        $ 3381 "bajar≔pose_add(get_actual_tcp_pose(), bajada_broca)"
        global bajar= pose_add ( get_actual_tcp_pose (), bajada_broca)
        $ 3382 "bajar" "breakAfter"
        movel(bajar, a=0.005, v=0.001)
        $ 3383 "subir≔pose_sub(get_actual_tcp_pose(), bajada_broca)"
        global subir= pose_sub ( get_actual_tcp_pose (), bajada_broca)
        $ 3384 "subir" "breakAfter"
        movel(subir, a=0.01, v=0.01)
        $ 3385 "bajada_broca≔pose_sub(bajada_broca, bajada)"
        global bajada_broca= pose_sub (bajada_broca, bajada)
        Loop_58 = Loop_58 + 1
      end
      $ 3386 "Direction: Base Z+"
      global move_thread_flag_3386=0
      thread move_thread_3386():
        enter_critical
        move_thread_flag_3386 = 1
        local towardsPos=calculate_point_to_move_towards(p[0.0,0.0,0.0,0.0,0.0,0.0], [0.0,0.0,1.0], 0.06)
        movel(towardsPos, a=0.035, v=0.03)
        move_thread_flag_3386 = 2
        exit_critical
      end
      move_thread_flag_3386 = 0
      move_thread_han_3386 = run move_thread_3386()
      while (True):
        sleep(1.0E-10)
        if (move_thread_flag_3386 > 1):
          join move_thread_han_3386
          $ 3387 "Until (distance)"
          break
        end
        sync()
      end
      $ 3388 "Set CO[1]=Apagar"
      set_configurable_digital_out(1, False)
      $ 3389 "barreno_actual≔barreno_actual+1"
      global barreno_actual=barreno_actual+1
      $ 3390 "If barreno_actual≥barrenos_menos1"
      if (barreno_actual >= barrenos_menos1):
        $ 3391 "cambiar_broca≔ True "
        global cambiar_broca=  True
      end
    end
    $ 3394 "Popup: Linea4 con chica Terminada!"
    popup("Linea4 con chica Terminada!", "Mensaje", False, False, blocking=True)
    $ 3395 "Broca_2"
    $ 3396 "Linea3"
    $ 3397 "Marcar_puntos"
    $ 3398 "MoveL"
    $ 3399 "Home3" "breakAfter"
    movel(Home3_p, a=0.5, v=0.1)
    $ 3400 "Linea3_A" "breakAfter"
    movel(Linea3_A_p, a=0.5, v=0.1)
    $ 3401 "Linea3_B" "breakAfter"
    movel(Linea3_B_p, a=0.5, v=0.1)
    $ 3402 "Linea3_C" "breakAfter"
    movel(Linea3_C_p, a=0.5, v=0.1)
    $ 3403 "Linea3_D" "breakAfter"
    movel(Linea3_D_p, a=0.5, v=0.1)
    $ 3404 "Linea3_E" "breakAfter"
    movel(Linea3_E_p, a=0.5, v=0.1)
    $ 3405 "Linea3_F" "breakAfter"
    movel(Linea3_F_p, a=0.5, v=0.1)
    $ 3406 "AB"
    $ 3407 "'desbaste_inicial'"
    # 'desbaste_inicial'
    $ 3408 "bajada_broca≔p[0,0,-0.012,0,0,0]"
    global bajada_broca=p[0,0,-0.012,0,0,0]
    $ 3409 "barrenos_menos1≔8"
    global barrenos_menos1=8
    $ 3410 "barreno_actual≔0"
    global barreno_actual=0
    $ 3411 "Loop barreno_actual≤barrenos_menos1"
    while (barreno_actual <= barrenos_menos1):
      $ 3412 "Perforacion"
      $ 3413 "MoveL"
      $ 3414 "internos≔interpolate_pose(Linea3_A, Linea3_B, barreno_actual/barrenos_menos1)"
      global internos= interpolate_pose (Linea3_A_p, Linea3_B_p, barreno_actual/barrenos_menos1)
      $ 3415 "internos" "breakAfter"
      movel(internos, a=0.5, v=0.1)
      $ 3416 "'desbaste_inicial'"
      # 'desbaste_inicial'
      $ 3417 "bajada_broca≔p[0,0,-0.012,0,0,0]"
      global bajada_broca=p[0,0,-0.012,0,0,0]
      $ 3418 "bajada≔p[0,0,0.012,0,0,0]"
      global bajada=p[0,0,0.012,0,0,0]
      $ 3419 "Direction: Base Z-"
      global move_thread_flag_3419=0
      thread move_thread_3419():
        enter_critical
        move_thread_flag_3419 = 1
        local towardsPos=calculate_point_to_move_towards(p[0.0,0.0,0.0,0.0,0.0,0.0], [0.0,0.0,-1.0], 0.076)
        movel(towardsPos, a=0.015, v=0.02)
        move_thread_flag_3419 = 2
        exit_critical
      end
      move_thread_flag_3419 = 0
      move_thread_han_3419 = run move_thread_3419()
      while (True):
        sleep(1.0E-10)
        if (move_thread_flag_3419 > 1):
          join move_thread_han_3419
          $ 3420 "Until (distance)"
          break
        end
        sync()
      end
      $ 3421 "Popup: punto contacto alanzdo"
      popup("punto contacto alanzdo", "Mensaje", False, False, blocking=True)
      $ 3422 "Direction: Base Z+"
      global move_thread_flag_3422=0
      thread move_thread_3422():
        enter_critical
        move_thread_flag_3422 = 1
        local towardsPos=calculate_point_to_move_towards(p[0.0,0.0,0.0,0.0,0.0,0.0], [0.0,0.0,1.0], 0.002)
        movel(towardsPos, a=0.005, v=0.003)
        move_thread_flag_3422 = 2
        exit_critical
      end
      move_thread_flag_3422 = 0
      move_thread_han_3422 = run move_thread_3422()
      while (True):
        sleep(1.0E-10)
        if (move_thread_flag_3422 > 1):
          join move_thread_han_3422
          $ 3423 "Until (distance)"
          break
        end
        sync()
      end
      $ 3424 "Wait: 0.3"
      sleep(0.3)
      $ 3425 "Set CO[1]=Encender"
      set_configurable_digital_out(1, True)
      $ 3426 "Wait: 0.3"
      sleep(0.3)
      $ 3427 "Loop 2 times"
      Loop_60 = 0
      while (Loop_60 < 2):
        $ 3428 "bajar≔pose_add(get_actual_tcp_pose(), bajada_broca)"
        global bajar= pose_add ( get_actual_tcp_pose (), bajada_broca)
        $ 3429 "bajar" "breakAfter"
        movel(bajar, a=0.005, v=0.001)
        $ 3430 "subir≔pose_sub(get_actual_tcp_pose(), bajada_broca)"
        global subir= pose_sub ( get_actual_tcp_pose (), bajada_broca)
        $ 3431 "subir" "breakAfter"
        movel(subir, a=0.01, v=0.01)
        $ 3432 "bajada_broca≔pose_sub(bajada_broca, bajada)"
        global bajada_broca= pose_sub (bajada_broca, bajada)
        Loop_60 = Loop_60 + 1
      end
      $ 3433 "Direction: Base Z+"
      global move_thread_flag_3433=0
      thread move_thread_3433():
        enter_critical
        move_thread_flag_3433 = 1
        local towardsPos=calculate_point_to_move_towards(p[0.0,0.0,0.0,0.0,0.0,0.0], [0.0,0.0,1.0], 0.06)
        movel(towardsPos, a=0.035, v=0.03)
        move_thread_flag_3433 = 2
        exit_critical
      end
      move_thread_flag_3433 = 0
      move_thread_han_3433 = run move_thread_3433()
      while (True):
        sleep(1.0E-10)
        if (move_thread_flag_3433 > 1):
          join move_thread_han_3433
          $ 3434 "Until (distance)"
          break
        end
        sync()
      end
      $ 3435 "Set CO[1]=Apagar"
      set_configurable_digital_out(1, False)
      $ 3436 "barreno_actual≔barreno_actual+1"
      global barreno_actual=barreno_actual+1
    end
    $ 3439 "CD"
    $ 3440 "'desbaste_inicial'"
    # 'desbaste_inicial'
    $ 3441 "bajada_broca≔p[0,0,-0.012,0,0,0]"
    global bajada_broca=p[0,0,-0.012,0,0,0]
    $ 3442 "barrenos_menos1≔8"
    global barrenos_menos1=8
    $ 3443 "barreno_actual≔0"
    global barreno_actual=0
    $ 3444 "Loop barreno_actual≤barrenos_menos1"
    while (barreno_actual <= barrenos_menos1):
      $ 3445 "Perforacion"
      $ 3446 "MoveL"
      $ 3447 "internos≔interpolate_pose(Linea3_C, Linea3_D, barreno_actual/barrenos_menos1)"
      global internos= interpolate_pose (Linea3_C_p, Linea3_D_p, barreno_actual/barrenos_menos1)
      $ 3448 "internos" "breakAfter"
      movel(internos, a=0.5, v=0.1)
      $ 3449 "'desbaste_inicial'"
      # 'desbaste_inicial'
      $ 3450 "bajada_broca≔p[0,0,-0.012,0,0,0]"
      global bajada_broca=p[0,0,-0.012,0,0,0]
      $ 3451 "bajada≔p[0,0,0.012,0,0,0]"
      global bajada=p[0,0,0.012,0,0,0]
      $ 3452 "Direction: Base Z-"
      global move_thread_flag_3452=0
      thread move_thread_3452():
        enter_critical
        move_thread_flag_3452 = 1
        local towardsPos=calculate_point_to_move_towards(p[0.0,0.0,0.0,0.0,0.0,0.0], [0.0,0.0,-1.0], 0.076)
        movel(towardsPos, a=0.015, v=0.02)
        move_thread_flag_3452 = 2
        exit_critical
      end
      move_thread_flag_3452 = 0
      move_thread_han_3452 = run move_thread_3452()
      while (True):
        sleep(1.0E-10)
        if (move_thread_flag_3452 > 1):
          join move_thread_han_3452
          $ 3453 "Until (distance)"
          break
        end
        sync()
      end
      $ 3454 "Popup: punto contacto alanzdo"
      popup("punto contacto alanzdo", "Mensaje", False, False, blocking=True)
      $ 3455 "Direction: Base Z+"
      global move_thread_flag_3455=0
      thread move_thread_3455():
        enter_critical
        move_thread_flag_3455 = 1
        local towardsPos=calculate_point_to_move_towards(p[0.0,0.0,0.0,0.0,0.0,0.0], [0.0,0.0,1.0], 0.002)
        movel(towardsPos, a=0.005, v=0.003)
        move_thread_flag_3455 = 2
        exit_critical
      end
      move_thread_flag_3455 = 0
      move_thread_han_3455 = run move_thread_3455()
      while (True):
        sleep(1.0E-10)
        if (move_thread_flag_3455 > 1):
          join move_thread_han_3455
          $ 3456 "Until (distance)"
          break
        end
        sync()
      end
      $ 3457 "Wait: 0.3"
      sleep(0.3)
      $ 3458 "Set CO[1]=Encender"
      set_configurable_digital_out(1, True)
      $ 3459 "Wait: 0.3"
      sleep(0.3)
      $ 3460 "Loop 2 times"
      Loop_64 = 0
      while (Loop_64 < 2):
        $ 3461 "bajar≔pose_add(get_actual_tcp_pose(), bajada_broca)"
        global bajar= pose_add ( get_actual_tcp_pose (), bajada_broca)
        $ 3462 "bajar" "breakAfter"
        movel(bajar, a=0.005, v=0.001)
        $ 3463 "subir≔pose_sub(get_actual_tcp_pose(), bajada_broca)"
        global subir= pose_sub ( get_actual_tcp_pose (), bajada_broca)
        $ 3464 "subir" "breakAfter"
        movel(subir, a=0.01, v=0.01)
        $ 3465 "bajada_broca≔pose_sub(bajada_broca, bajada)"
        global bajada_broca= pose_sub (bajada_broca, bajada)
        Loop_64 = Loop_64 + 1
      end
      $ 3466 "Direction: Base Z+"
      global move_thread_flag_3466=0
      thread move_thread_3466():
        enter_critical
        move_thread_flag_3466 = 1
        local towardsPos=calculate_point_to_move_towards(p[0.0,0.0,0.0,0.0,0.0,0.0], [0.0,0.0,1.0], 0.06)
        movel(towardsPos, a=0.035, v=0.03)
        move_thread_flag_3466 = 2
        exit_critical
      end
      move_thread_flag_3466 = 0
      move_thread_han_3466 = run move_thread_3466()
      while (True):
        sleep(1.0E-10)
        if (move_thread_flag_3466 > 1):
          join move_thread_han_3466
          $ 3467 "Until (distance)"
          break
        end
        sync()
      end
      $ 3468 "Set CO[1]=Apagar"
      set_configurable_digital_out(1, False)
      $ 3469 "barreno_actual≔barreno_actual+1"
      global barreno_actual=barreno_actual+1
    end
    $ 3472 "EF"
    $ 3473 "'desbaste_inicial'"
    # 'desbaste_inicial'
    $ 3474 "bajada_broca≔p[0,0,-0.012,0,0,0]"
    global bajada_broca=p[0,0,-0.012,0,0,0]
    $ 3475 "barrenos_menos1≔8"
    global barrenos_menos1=8
    $ 3476 "barreno_actual≔0"
    global barreno_actual=0
    $ 3477 "Loop barreno_actual≤barrenos_menos1"
    while (barreno_actual <= barrenos_menos1):
      $ 3478 "Perforacion"
      $ 3479 "MoveL"
      $ 3480 "internos≔interpolate_pose(Linea3_E, Linea3_F, barreno_actual/barrenos_menos1)"
      global internos= interpolate_pose (Linea3_E_p, Linea3_F_p, barreno_actual/barrenos_menos1)
      $ 3481 "internos" "breakAfter"
      movel(internos, a=0.5, v=0.1)
      $ 3482 "'desbaste_inicial'"
      # 'desbaste_inicial'
      $ 3483 "bajada_broca≔p[0,0,-0.012,0,0,0]"
      global bajada_broca=p[0,0,-0.012,0,0,0]
      $ 3484 "bajada≔p[0,0,0.012,0,0,0]"
      global bajada=p[0,0,0.012,0,0,0]
      $ 3485 "Direction: Base Z-"
      global move_thread_flag_3485=0
      thread move_thread_3485():
        enter_critical
        move_thread_flag_3485 = 1
        local towardsPos=calculate_point_to_move_towards(p[0.0,0.0,0.0,0.0,0.0,0.0], [0.0,0.0,-1.0], 0.076)
        movel(towardsPos, a=0.015, v=0.02)
        move_thread_flag_3485 = 2
        exit_critical
      end
      move_thread_flag_3485 = 0
      move_thread_han_3485 = run move_thread_3485()
      while (True):
        sleep(1.0E-10)
        if (move_thread_flag_3485 > 1):
          join move_thread_han_3485
          $ 3486 "Until (distance)"
          break
        end
        sync()
      end
      $ 3487 "Popup: punto contacto alanzdo"
      popup("punto contacto alanzdo", "Mensaje", False, False, blocking=True)
      $ 3488 "Direction: Base Z+"
      global move_thread_flag_3488=0
      thread move_thread_3488():
        enter_critical
        move_thread_flag_3488 = 1
        local towardsPos=calculate_point_to_move_towards(p[0.0,0.0,0.0,0.0,0.0,0.0], [0.0,0.0,1.0], 0.002)
        movel(towardsPos, a=0.005, v=0.003)
        move_thread_flag_3488 = 2
        exit_critical
      end
      move_thread_flag_3488 = 0
      move_thread_han_3488 = run move_thread_3488()
      while (True):
        sleep(1.0E-10)
        if (move_thread_flag_3488 > 1):
          join move_thread_han_3488
          $ 3489 "Until (distance)"
          break
        end
        sync()
      end
      $ 3490 "Wait: 0.3"
      sleep(0.3)
      $ 3491 "Set CO[1]=Encender"
      set_configurable_digital_out(1, True)
      $ 3492 "Wait: 0.3"
      sleep(0.3)
      $ 3493 "Loop 2 times"
      Loop_68 = 0
      while (Loop_68 < 2):
        $ 3494 "bajar≔pose_add(get_actual_tcp_pose(), bajada_broca)"
        global bajar= pose_add ( get_actual_tcp_pose (), bajada_broca)
        $ 3495 "bajar" "breakAfter"
        movel(bajar, a=0.005, v=0.001)
        $ 3496 "subir≔pose_sub(get_actual_tcp_pose(), bajada_broca)"
        global subir= pose_sub ( get_actual_tcp_pose (), bajada_broca)
        $ 3497 "subir" "breakAfter"
        movel(subir, a=0.01, v=0.01)
        $ 3498 "bajada_broca≔pose_sub(bajada_broca, bajada)"
        global bajada_broca= pose_sub (bajada_broca, bajada)
        Loop_68 = Loop_68 + 1
      end
      $ 3499 "Direction: Base Z+"
      global move_thread_flag_3499=0
      thread move_thread_3499():
        enter_critical
        move_thread_flag_3499 = 1
        local towardsPos=calculate_point_to_move_towards(p[0.0,0.0,0.0,0.0,0.0,0.0], [0.0,0.0,1.0], 0.06)
        movel(towardsPos, a=0.035, v=0.03)
        move_thread_flag_3499 = 2
        exit_critical
      end
      move_thread_flag_3499 = 0
      move_thread_han_3499 = run move_thread_3499()
      while (True):
        sleep(1.0E-10)
        if (move_thread_flag_3499 > 1):
          join move_thread_han_3499
          $ 3500 "Until (distance)"
          break
        end
        sync()
      end
      $ 3501 "Set CO[1]=Apagar"
      set_configurable_digital_out(1, False)
      $ 3502 "barreno_actual≔barreno_actual+1"
      global barreno_actual=barreno_actual+1
    end
    $ 3505 "Popup: Linea3 con media Terminada!"
    popup("Linea3 con media Terminada!", "Mensaje", False, False, blocking=True)
    $ 3506 "Linea4"
    $ 3507 "Marcar_puntos"
    $ 3508 "MoveL"
    $ 3509 "Home3" "breakAfter"
    movel(Home3_p, a=0.5, v=0.1)
    $ 3510 "Linea4_A" "breakAfter"
    movel(Linea4_A_p, a=0.5, v=0.1)
    $ 3511 "Linea4_B" "breakAfter"
    movel(Linea4_B_p, a=0.5, v=0.1)
    $ 3512 "Linea4_C" "breakAfter"
    movel(Linea4_C_p, a=0.5, v=0.1)
    $ 3513 "Linea4_D" "breakAfter"
    movel(Linea4_D_p, a=0.5, v=0.1)
    $ 3514 "Linea4_E" "breakAfter"
    movel(Linea4_E_p, a=0.5, v=0.1)
    $ 3515 "Linea4_F" "breakAfter"
    movel(Linea4_F_p, a=0.5, v=0.1)
    $ 3516 "AB"
    $ 3517 "'desbaste_inicial'"
    # 'desbaste_inicial'
    $ 3518 "bajada_broca≔p[0,0,-0.012,0,0,0]"
    global bajada_broca=p[0,0,-0.012,0,0,0]
    $ 3519 "barrenos_menos1≔8"
    global barrenos_menos1=8
    $ 3520 "barreno_actual≔0"
    global barreno_actual=0
    $ 3521 "Loop barreno_actual≤barrenos_menos1"
    while (barreno_actual <= barrenos_menos1):
      $ 3522 "Perforacion"
      $ 3523 "MoveL"
      $ 3524 "internos≔interpolate_pose(Linea4_A, Linea4_B, barreno_actual/barrenos_menos1)"
      global internos= interpolate_pose (Linea4_A_p, Linea4_B_p, barreno_actual/barrenos_menos1)
      $ 3525 "internos" "breakAfter"
      movel(internos, a=0.5, v=0.1)
      $ 3526 "'desbaste_inicial'"
      # 'desbaste_inicial'
      $ 3527 "bajada_broca≔p[0,0,-0.012,0,0,0]"
      global bajada_broca=p[0,0,-0.012,0,0,0]
      $ 3528 "bajada≔p[0,0,0.012,0,0,0]"
      global bajada=p[0,0,0.012,0,0,0]
      $ 3529 "Direction: Base Z-"
      global move_thread_flag_3529=0
      thread move_thread_3529():
        enter_critical
        move_thread_flag_3529 = 1
        local towardsPos=calculate_point_to_move_towards(p[0.0,0.0,0.0,0.0,0.0,0.0], [0.0,0.0,-1.0], 0.073)
        movel(towardsPos, a=0.015, v=0.02)
        move_thread_flag_3529 = 2
        exit_critical
      end
      move_thread_flag_3529 = 0
      move_thread_han_3529 = run move_thread_3529()
      while (True):
        sleep(1.0E-10)
        if (move_thread_flag_3529 > 1):
          join move_thread_han_3529
          $ 3530 "Until (distance)"
          break
        end
        sync()
      end
      $ 3531 "Popup: punto contacto alanzdo"
      popup("punto contacto alanzdo", "Mensaje", False, False, blocking=True)
      $ 3532 "Direction: Base Z+"
      global move_thread_flag_3532=0
      thread move_thread_3532():
        enter_critical
        move_thread_flag_3532 = 1
        local towardsPos=calculate_point_to_move_towards(p[0.0,0.0,0.0,0.0,0.0,0.0], [0.0,0.0,1.0], 0.002)
        movel(towardsPos, a=0.005, v=0.003)
        move_thread_flag_3532 = 2
        exit_critical
      end
      move_thread_flag_3532 = 0
      move_thread_han_3532 = run move_thread_3532()
      while (True):
        sleep(1.0E-10)
        if (move_thread_flag_3532 > 1):
          join move_thread_han_3532
          $ 3533 "Until (distance)"
          break
        end
        sync()
      end
      $ 3534 "Wait: 0.3"
      sleep(0.3)
      $ 3535 "Set CO[1]=Encender"
      set_configurable_digital_out(1, True)
      $ 3536 "Wait: 0.3"
      sleep(0.3)
      $ 3537 "Loop 2 times"
      Loop_72 = 0
      while (Loop_72 < 2):
        $ 3538 "bajar≔pose_add(get_actual_tcp_pose(), bajada_broca)"
        global bajar= pose_add ( get_actual_tcp_pose (), bajada_broca)
        $ 3539 "bajar" "breakAfter"
        movel(bajar, a=0.005, v=0.001)
        $ 3540 "subir≔pose_sub(get_actual_tcp_pose(), bajada_broca)"
        global subir= pose_sub ( get_actual_tcp_pose (), bajada_broca)
        $ 3541 "subir" "breakAfter"
        movel(subir, a=0.01, v=0.01)
        $ 3542 "bajada_broca≔pose_sub(bajada_broca, bajada)"
        global bajada_broca= pose_sub (bajada_broca, bajada)
        Loop_72 = Loop_72 + 1
      end
      $ 3543 "Direction: Base Z+"
      global move_thread_flag_3543=0
      thread move_thread_3543():
        enter_critical
        move_thread_flag_3543 = 1
        local towardsPos=calculate_point_to_move_towards(p[0.0,0.0,0.0,0.0,0.0,0.0], [0.0,0.0,1.0], 0.06)
        movel(towardsPos, a=0.035, v=0.03)
        move_thread_flag_3543 = 2
        exit_critical
      end
      move_thread_flag_3543 = 0
      move_thread_han_3543 = run move_thread_3543()
      while (True):
        sleep(1.0E-10)
        if (move_thread_flag_3543 > 1):
          join move_thread_han_3543
          $ 3544 "Until (distance)"
          break
        end
        sync()
      end
      $ 3545 "Set CO[1]=Apagar"
      set_configurable_digital_out(1, False)
      $ 3546 "barreno_actual≔barreno_actual+1"
      global barreno_actual=barreno_actual+1
    end
    $ 3549 "CD"
    $ 3550 "'desbaste_inicial'"
    # 'desbaste_inicial'
    $ 3551 "bajada_broca≔p[0,0,-0.012,0,0,0]"
    global bajada_broca=p[0,0,-0.012,0,0,0]
    $ 3552 "barrenos_menos1≔8"
    global barrenos_menos1=8
    $ 3553 "barreno_actual≔0"
    global barreno_actual=0
    $ 3554 "Loop barreno_actual≤barrenos_menos1"
    while (barreno_actual <= barrenos_menos1):
      $ 3555 "Perforacion"
      $ 3556 "MoveL"
      $ 3557 "internos≔interpolate_pose(Linea4_C, Linea4_D, barreno_actual/barrenos_menos1)"
      global internos= interpolate_pose (Linea4_C_p, Linea4_D_p, barreno_actual/barrenos_menos1)
      $ 3558 "internos" "breakAfter"
      movel(internos, a=0.5, v=0.1)
      $ 3559 "'desbaste_inicial'"
      # 'desbaste_inicial'
      $ 3560 "bajada_broca≔p[0,0,-0.012,0,0,0]"
      global bajada_broca=p[0,0,-0.012,0,0,0]
      $ 3561 "bajada≔p[0,0,0.012,0,0,0]"
      global bajada=p[0,0,0.012,0,0,0]
      $ 3562 "Direction: Base Z-"
      global move_thread_flag_3562=0
      thread move_thread_3562():
        enter_critical
        move_thread_flag_3562 = 1
        local towardsPos=calculate_point_to_move_towards(p[0.0,0.0,0.0,0.0,0.0,0.0], [0.0,0.0,-1.0], 0.073)
        movel(towardsPos, a=0.015, v=0.02)
        move_thread_flag_3562 = 2
        exit_critical
      end
      move_thread_flag_3562 = 0
      move_thread_han_3562 = run move_thread_3562()
      while (True):
        sleep(1.0E-10)
        if (move_thread_flag_3562 > 1):
          join move_thread_han_3562
          $ 3563 "Until (distance)"
          break
        end
        sync()
      end
      $ 3564 "Popup: punto contacto alanzdo"
      popup("punto contacto alanzdo", "Mensaje", False, False, blocking=True)
      $ 3565 "Direction: Base Z+"
      global move_thread_flag_3565=0
      thread move_thread_3565():
        enter_critical
        move_thread_flag_3565 = 1
        local towardsPos=calculate_point_to_move_towards(p[0.0,0.0,0.0,0.0,0.0,0.0], [0.0,0.0,1.0], 0.002)
        movel(towardsPos, a=0.005, v=0.003)
        move_thread_flag_3565 = 2
        exit_critical
      end
      move_thread_flag_3565 = 0
      move_thread_han_3565 = run move_thread_3565()
      while (True):
        sleep(1.0E-10)
        if (move_thread_flag_3565 > 1):
          join move_thread_han_3565
          $ 3566 "Until (distance)"
          break
        end
        sync()
      end
      $ 3567 "Wait: 0.3"
      sleep(0.3)
      $ 3568 "Set CO[1]=Encender"
      set_configurable_digital_out(1, True)
      $ 3569 "Wait: 0.3"
      sleep(0.3)
      $ 3570 "Loop 2 times"
      Loop_77 = 0
      while (Loop_77 < 2):
        $ 3571 "bajar≔pose_add(get_actual_tcp_pose(), bajada_broca)"
        global bajar= pose_add ( get_actual_tcp_pose (), bajada_broca)
        $ 3572 "bajar" "breakAfter"
        movel(bajar, a=0.005, v=0.001)
        $ 3573 "subir≔pose_sub(get_actual_tcp_pose(), bajada_broca)"
        global subir= pose_sub ( get_actual_tcp_pose (), bajada_broca)
        $ 3574 "subir" "breakAfter"
        movel(subir, a=0.01, v=0.01)
        $ 3575 "bajada_broca≔pose_sub(bajada_broca, bajada)"
        global bajada_broca= pose_sub (bajada_broca, bajada)
        Loop_77 = Loop_77 + 1
      end
      $ 3576 "Direction: Base Z+"
      global move_thread_flag_3576=0
      thread move_thread_3576():
        enter_critical
        move_thread_flag_3576 = 1
        local towardsPos=calculate_point_to_move_towards(p[0.0,0.0,0.0,0.0,0.0,0.0], [0.0,0.0,1.0], 0.06)
        movel(towardsPos, a=0.035, v=0.03)
        move_thread_flag_3576 = 2
        exit_critical
      end
      move_thread_flag_3576 = 0
      move_thread_han_3576 = run move_thread_3576()
      while (True):
        sleep(1.0E-10)
        if (move_thread_flag_3576 > 1):
          join move_thread_han_3576
          $ 3577 "Until (distance)"
          break
        end
        sync()
      end
      $ 3578 "Set CO[1]=Apagar"
      set_configurable_digital_out(1, False)
      $ 3579 "barreno_actual≔barreno_actual+1"
      global barreno_actual=barreno_actual+1
    end
    $ 3582 "EF"
    $ 3583 "'desbaste_inicial'"
    # 'desbaste_inicial'
    $ 3584 "bajada_broca≔p[0,0,-0.012,0,0,0]"
    global bajada_broca=p[0,0,-0.012,0,0,0]
    $ 3585 "barrenos_menos1≔8"
    global barrenos_menos1=8
    $ 3586 "barreno_actual≔0"
    global barreno_actual=0
    $ 3587 "Loop barreno_actual≤barrenos_menos1"
    while (barreno_actual <= barrenos_menos1):
      $ 3588 "Perforacion"
      $ 3589 "MoveL"
      $ 3590 "internos≔interpolate_pose(Linea4_E, Linea4_F, barreno_actual/barrenos_menos1)"
      global internos= interpolate_pose (Linea4_E_p, Linea4_F_p, barreno_actual/barrenos_menos1)
      $ 3591 "internos" "breakAfter"
      movel(internos, a=0.5, v=0.1)
      $ 3592 "'desbaste_inicial'"
      # 'desbaste_inicial'
      $ 3593 "bajada_broca≔p[0,0,-0.012,0,0,0]"
      global bajada_broca=p[0,0,-0.012,0,0,0]
      $ 3594 "bajada≔p[0,0,0.012,0,0,0]"
      global bajada=p[0,0,0.012,0,0,0]
      $ 3595 "Direction: Base Z-"
      global move_thread_flag_3595=0
      thread move_thread_3595():
        enter_critical
        move_thread_flag_3595 = 1
        local towardsPos=calculate_point_to_move_towards(p[0.0,0.0,0.0,0.0,0.0,0.0], [0.0,0.0,-1.0], 0.073)
        movel(towardsPos, a=0.015, v=0.02)
        move_thread_flag_3595 = 2
        exit_critical
      end
      move_thread_flag_3595 = 0
      move_thread_han_3595 = run move_thread_3595()
      while (True):
        sleep(1.0E-10)
        if (move_thread_flag_3595 > 1):
          join move_thread_han_3595
          $ 3596 "Until (distance)"
          break
        end
        sync()
      end
      $ 3597 "Popup: punto contacto alanzdo"
      popup("punto contacto alanzdo", "Mensaje", False, False, blocking=True)
      $ 3598 "Direction: Base Z+"
      global move_thread_flag_3598=0
      thread move_thread_3598():
        enter_critical
        move_thread_flag_3598 = 1
        local towardsPos=calculate_point_to_move_towards(p[0.0,0.0,0.0,0.0,0.0,0.0], [0.0,0.0,1.0], 0.002)
        movel(towardsPos, a=0.005, v=0.003)
        move_thread_flag_3598 = 2
        exit_critical
      end
      move_thread_flag_3598 = 0
      move_thread_han_3598 = run move_thread_3598()
      while (True):
        sleep(1.0E-10)
        if (move_thread_flag_3598 > 1):
          join move_thread_han_3598
          $ 3599 "Until (distance)"
          break
        end
        sync()
      end
      $ 3600 "Wait: 0.3"
      sleep(0.3)
      $ 3601 "Set CO[1]=Encender"
      set_configurable_digital_out(1, True)
      $ 3602 "Wait: 0.3"
      sleep(0.3)
      $ 3603 "Loop 2 times"
      Loop_81 = 0
      while (Loop_81 < 2):
        $ 3604 "bajar≔pose_add(get_actual_tcp_pose(), bajada_broca)"
        global bajar= pose_add ( get_actual_tcp_pose (), bajada_broca)
        $ 3605 "bajar" "breakAfter"
        movel(bajar, a=0.005, v=0.001)
        $ 3606 "subir≔pose_sub(get_actual_tcp_pose(), bajada_broca)"
        global subir= pose_sub ( get_actual_tcp_pose (), bajada_broca)
        $ 3607 "subir" "breakAfter"
        movel(subir, a=0.01, v=0.01)
        $ 3608 "bajada_broca≔pose_sub(bajada_broca, bajada)"
        global bajada_broca= pose_sub (bajada_broca, bajada)
        Loop_81 = Loop_81 + 1
      end
      $ 3609 "Direction: Base Z+"
      global move_thread_flag_3609=0
      thread move_thread_3609():
        enter_critical
        move_thread_flag_3609 = 1
        local towardsPos=calculate_point_to_move_towards(p[0.0,0.0,0.0,0.0,0.0,0.0], [0.0,0.0,1.0], 0.06)
        movel(towardsPos, a=0.035, v=0.03)
        move_thread_flag_3609 = 2
        exit_critical
      end
      move_thread_flag_3609 = 0
      move_thread_han_3609 = run move_thread_3609()
      while (True):
        sleep(1.0E-10)
        if (move_thread_flag_3609 > 1):
          join move_thread_han_3609
          $ 3610 "Until (distance)"
          break
        end
        sync()
      end
      $ 3611 "Set CO[1]=Apagar"
      set_configurable_digital_out(1, False)
      $ 3612 "barreno_actual≔barreno_actual+1"
      global barreno_actual=barreno_actual+1
      $ 3613 "If barreno_actual≥barrenos_menos1"
      if (barreno_actual >= barrenos_menos1):
        $ 3614 "cambiar_broca≔ True "
        global cambiar_broca=  True
      end
    end
    $ 3617 "Popup: Linea4 con media Terminada!"
    popup("Linea4 con media Terminada!", "Mensaje", False, False, blocking=True)
    $ 3618 "Broca_3"
    $ 3619 "Linea3"
    $ 3620 "Marcar_puntos"
    $ 3621 "MoveL"
    $ 3622 "Home3" "breakAfter"
    movel(Home3_p, a=0.5, v=0.1)
    $ 3623 "Linea3_A" "breakAfter"
    movel(Linea3_A_p, a=0.5, v=0.1)
    $ 3624 "Linea3_B" "breakAfter"
    movel(Linea3_B_p, a=0.5, v=0.1)
    $ 3625 "Linea3_C" "breakAfter"
    movel(Linea3_C_p, a=0.5, v=0.1)
    $ 3626 "Linea3_D" "breakAfter"
    movel(Linea3_D_p, a=0.5, v=0.1)
    $ 3627 "Linea3_E" "breakAfter"
    movel(Linea3_E_p, a=0.5, v=0.1)
    $ 3628 "Linea3_F" "breakAfter"
    movel(Linea3_F_p, a=0.5, v=0.1)
    $ 3629 "AB"
    $ 3630 "'desbaste_inicial'"
    # 'desbaste_inicial'
    $ 3631 "bajada_broca≔p[0,0,-0.024,0,0,0]"
    global bajada_broca=p[0,0,-0.024,0,0,0]
    $ 3632 "barrenos_menos1≔8"
    global barrenos_menos1=8
    $ 3633 "barreno_actual≔0"
    global barreno_actual=0
    $ 3634 "Loop barreno_actual≤barrenos_menos1"
    while (barreno_actual <= barrenos_menos1):
      $ 3635 "Perforacion"
      $ 3636 "MoveL"
      $ 3637 "internos≔interpolate_pose(Linea3_A, Linea3_B, barreno_actual/barrenos_menos1)"
      global internos= interpolate_pose (Linea3_A_p, Linea3_B_p, barreno_actual/barrenos_menos1)
      $ 3638 "internos" "breakAfter"
      movel(internos, a=0.5, v=0.1)
      $ 3639 "'desbaste_inicial'"
      # 'desbaste_inicial'
      $ 3640 "bajada_broca≔p[0,0,-0.024,0,0,0]"
      global bajada_broca=p[0,0,-0.024,0,0,0]
      $ 3641 "bajada≔p[0,0,0.024,0,0,0]"
      global bajada=p[0,0,0.024,0,0,0]
      $ 3642 "Direction: Base Z-"
      global move_thread_flag_3642=0
      thread move_thread_3642():
        enter_critical
        move_thread_flag_3642 = 1
        local towardsPos=calculate_point_to_move_towards(p[0.0,0.0,0.0,0.0,0.0,0.0], [0.0,0.0,-1.0], 0.076)
        movel(towardsPos, a=0.015, v=0.02)
        move_thread_flag_3642 = 2
        exit_critical
      end
      move_thread_flag_3642 = 0
      move_thread_han_3642 = run move_thread_3642()
      while (True):
        sleep(1.0E-10)
        if (move_thread_flag_3642 > 1):
          join move_thread_han_3642
          $ 3643 "Until (distance)"
          break
        end
        sync()
      end
      $ 3644 "Popup: punto contacto alanzdo"
      popup("punto contacto alanzdo", "Mensaje", False, False, blocking=True)
      $ 3645 "Direction: Base Z+"
      global move_thread_flag_3645=0
      thread move_thread_3645():
        enter_critical
        move_thread_flag_3645 = 1
        local towardsPos=calculate_point_to_move_towards(p[0.0,0.0,0.0,0.0,0.0,0.0], [0.0,0.0,1.0], 0.002)
        movel(towardsPos, a=0.005, v=0.003)
        move_thread_flag_3645 = 2
        exit_critical
      end
      move_thread_flag_3645 = 0
      move_thread_han_3645 = run move_thread_3645()
      while (True):
        sleep(1.0E-10)
        if (move_thread_flag_3645 > 1):
          join move_thread_han_3645
          $ 3646 "Until (distance)"
          break
        end
        sync()
      end
      $ 3647 "Wait: 0.3"
      sleep(0.3)
      $ 3648 "Set CO[1]=Encender"
      set_configurable_digital_out(1, True)
      $ 3649 "Wait: 0.3"
      sleep(0.3)
      $ 3650 "Loop 1 times"
      Loop_86 = 0
      while (Loop_86 < 1):
        $ 3651 "bajar≔pose_add(get_actual_tcp_pose(), bajada_broca)"
        global bajar= pose_add ( get_actual_tcp_pose (), bajada_broca)
        $ 3652 "bajar" "breakAfter"
        movel(bajar, a=0.005, v=0.001)
        $ 3653 "subir≔pose_sub(get_actual_tcp_pose(), bajada_broca)"
        global subir= pose_sub ( get_actual_tcp_pose (), bajada_broca)
        $ 3654 "subir" "breakAfter"
        movel(subir, a=0.01, v=0.01)
        $ 3655 "bajada_broca≔pose_sub(bajada_broca, bajada)"
        global bajada_broca= pose_sub (bajada_broca, bajada)
        Loop_86 = Loop_86 + 1
      end
      $ 3656 "Direction: Base Z+"
      global move_thread_flag_3656=0
      thread move_thread_3656():
        enter_critical
        move_thread_flag_3656 = 1
        local towardsPos=calculate_point_to_move_towards(p[0.0,0.0,0.0,0.0,0.0,0.0], [0.0,0.0,1.0], 0.06)
        movel(towardsPos, a=0.035, v=0.03)
        move_thread_flag_3656 = 2
        exit_critical
      end
      move_thread_flag_3656 = 0
      move_thread_han_3656 = run move_thread_3656()
      while (True):
        sleep(1.0E-10)
        if (move_thread_flag_3656 > 1):
          join move_thread_han_3656
          $ 3657 "Until (distance)"
          break
        end
        sync()
      end
      $ 3658 "Set CO[1]=Apagar"
      set_configurable_digital_out(1, False)
      $ 3659 "barreno_actual≔barreno_actual+1"
      global barreno_actual=barreno_actual+1
    end
    $ 3662 "CD"
    $ 3663 "'desbaste_inicial'"
    # 'desbaste_inicial'
    $ 3664 "bajada_broca≔p[0,0,-0.024,0,0,0]"
    global bajada_broca=p[0,0,-0.024,0,0,0]
    $ 3665 "barrenos_menos1≔8"
    global barrenos_menos1=8
    $ 3666 "barreno_actual≔0"
    global barreno_actual=0
    $ 3667 "Loop barreno_actual≤barrenos_menos1"
    while (barreno_actual <= barrenos_menos1):
      $ 3668 "Perforacion"
      $ 3669 "MoveL"
      $ 3670 "internos≔interpolate_pose(Linea3_C, Linea3_D, barreno_actual/barrenos_menos1)"
      global internos= interpolate_pose (Linea3_C_p, Linea3_D_p, barreno_actual/barrenos_menos1)
      $ 3671 "internos" "breakAfter"
      movel(internos, a=0.5, v=0.1)
      $ 3672 "'desbaste_inicial'"
      # 'desbaste_inicial'
      $ 3673 "bajada_broca≔p[0,0,-0.024,0,0,0]"
      global bajada_broca=p[0,0,-0.024,0,0,0]
      $ 3674 "bajada≔p[0,0,0.024,0,0,0]"
      global bajada=p[0,0,0.024,0,0,0]
      $ 3675 "Direction: Base Z-"
      global move_thread_flag_3675=0
      thread move_thread_3675():
        enter_critical
        move_thread_flag_3675 = 1
        local towardsPos=calculate_point_to_move_towards(p[0.0,0.0,0.0,0.0,0.0,0.0], [0.0,0.0,-1.0], 0.076)
        movel(towardsPos, a=0.015, v=0.02)
        move_thread_flag_3675 = 2
        exit_critical
      end
      move_thread_flag_3675 = 0
      move_thread_han_3675 = run move_thread_3675()
      while (True):
        sleep(1.0E-10)
        if (move_thread_flag_3675 > 1):
          join move_thread_han_3675
          $ 3676 "Until (distance)"
          break
        end
        sync()
      end
      $ 3677 "Popup: punto contacto alanzdo"
      popup("punto contacto alanzdo", "Mensaje", False, False, blocking=True)
      $ 3678 "Direction: Base Z+"
      global move_thread_flag_3678=0
      thread move_thread_3678():
        enter_critical
        move_thread_flag_3678 = 1
        local towardsPos=calculate_point_to_move_towards(p[0.0,0.0,0.0,0.0,0.0,0.0], [0.0,0.0,1.0], 0.002)
        movel(towardsPos, a=0.005, v=0.003)
        move_thread_flag_3678 = 2
        exit_critical
      end
      move_thread_flag_3678 = 0
      move_thread_han_3678 = run move_thread_3678()
      while (True):
        sleep(1.0E-10)
        if (move_thread_flag_3678 > 1):
          join move_thread_han_3678
          $ 3679 "Until (distance)"
          break
        end
        sync()
      end
      $ 3680 "Wait: 0.3"
      sleep(0.3)
      $ 3681 "Set CO[1]=Encender"
      set_configurable_digital_out(1, True)
      $ 3682 "Wait: 0.3"
      sleep(0.3)
      $ 3683 "Loop 1 times"
      Loop_91 = 0
      while (Loop_91 < 1):
        $ 3684 "bajar≔pose_add(get_actual_tcp_pose(), bajada_broca)"
        global bajar= pose_add ( get_actual_tcp_pose (), bajada_broca)
        $ 3685 "bajar" "breakAfter"
        movel(bajar, a=0.005, v=0.001)
        $ 3686 "subir≔pose_sub(get_actual_tcp_pose(), bajada_broca)"
        global subir= pose_sub ( get_actual_tcp_pose (), bajada_broca)
        $ 3687 "subir" "breakAfter"
        movel(subir, a=0.01, v=0.01)
        $ 3688 "bajada_broca≔pose_sub(bajada_broca, bajada)"
        global bajada_broca= pose_sub (bajada_broca, bajada)
        Loop_91 = Loop_91 + 1
      end
      $ 3689 "Direction: Base Z+"
      global move_thread_flag_3689=0
      thread move_thread_3689():
        enter_critical
        move_thread_flag_3689 = 1
        local towardsPos=calculate_point_to_move_towards(p[0.0,0.0,0.0,0.0,0.0,0.0], [0.0,0.0,1.0], 0.06)
        movel(towardsPos, a=0.035, v=0.03)
        move_thread_flag_3689 = 2
        exit_critical
      end
      move_thread_flag_3689 = 0
      move_thread_han_3689 = run move_thread_3689()
      while (True):
        sleep(1.0E-10)
        if (move_thread_flag_3689 > 1):
          join move_thread_han_3689
          $ 3690 "Until (distance)"
          break
        end
        sync()
      end
      $ 3691 "Set CO[1]=Apagar"
      set_configurable_digital_out(1, False)
      $ 3692 "barreno_actual≔barreno_actual+1"
      global barreno_actual=barreno_actual+1
    end
    $ 3695 "EF"
    $ 3696 "'desbaste_inicial'"
    # 'desbaste_inicial'
    $ 3697 "bajada_broca≔p[0,0,-0.024,0,0,0]"
    global bajada_broca=p[0,0,-0.024,0,0,0]
    $ 3698 "barrenos_menos1≔8"
    global barrenos_menos1=8
    $ 3699 "barreno_actual≔0"
    global barreno_actual=0
    $ 3700 "Loop barreno_actual≤barrenos_menos1"
    while (barreno_actual <= barrenos_menos1):
      $ 3701 "Perforacion"
      $ 3702 "MoveL"
      $ 3703 "internos≔interpolate_pose(Linea3_E, Linea3_F, barreno_actual/barrenos_menos1)"
      global internos= interpolate_pose (Linea3_E_p, Linea3_F_p, barreno_actual/barrenos_menos1)
      $ 3704 "internos" "breakAfter"
      movel(internos, a=0.5, v=0.1)
      $ 3705 "'desbaste_inicial'"
      # 'desbaste_inicial'
      $ 3706 "bajada_broca≔p[0,0,-0.024,0,0,0]"
      global bajada_broca=p[0,0,-0.024,0,0,0]
      $ 3707 "bajada≔p[0,0,0.024,0,0,0]"
      global bajada=p[0,0,0.024,0,0,0]
      $ 3708 "Direction: Base Z-"
      global move_thread_flag_3708=0
      thread move_thread_3708():
        enter_critical
        move_thread_flag_3708 = 1
        local towardsPos=calculate_point_to_move_towards(p[0.0,0.0,0.0,0.0,0.0,0.0], [0.0,0.0,-1.0], 0.076)
        movel(towardsPos, a=0.015, v=0.02)
        move_thread_flag_3708 = 2
        exit_critical
      end
      move_thread_flag_3708 = 0
      move_thread_han_3708 = run move_thread_3708()
      while (True):
        sleep(1.0E-10)
        if (move_thread_flag_3708 > 1):
          join move_thread_han_3708
          $ 3709 "Until (distance)"
          break
        end
        sync()
      end
      $ 3710 "Popup: punto contacto alanzdo"
      popup("punto contacto alanzdo", "Mensaje", False, False, blocking=True)
      $ 3711 "Direction: Base Z+"
      global move_thread_flag_3711=0
      thread move_thread_3711():
        enter_critical
        move_thread_flag_3711 = 1
        local towardsPos=calculate_point_to_move_towards(p[0.0,0.0,0.0,0.0,0.0,0.0], [0.0,0.0,1.0], 0.002)
        movel(towardsPos, a=0.005, v=0.003)
        move_thread_flag_3711 = 2
        exit_critical
      end
      move_thread_flag_3711 = 0
      move_thread_han_3711 = run move_thread_3711()
      while (True):
        sleep(1.0E-10)
        if (move_thread_flag_3711 > 1):
          join move_thread_han_3711
          $ 3712 "Until (distance)"
          break
        end
        sync()
      end
      $ 3713 "Wait: 0.3"
      sleep(0.3)
      $ 3714 "Set CO[1]=Encender"
      set_configurable_digital_out(1, True)
      $ 3715 "Wait: 0.3"
      sleep(0.3)
      $ 3716 "Loop 1 times"
      Loop_100 = 0
      while (Loop_100 < 1):
        $ 3717 "bajar≔pose_add(get_actual_tcp_pose(), bajada_broca)"
        global bajar= pose_add ( get_actual_tcp_pose (), bajada_broca)
        $ 3718 "bajar" "breakAfter"
        movel(bajar, a=0.005, v=0.001)
        $ 3719 "subir≔pose_sub(get_actual_tcp_pose(), bajada_broca)"
        global subir= pose_sub ( get_actual_tcp_pose (), bajada_broca)
        $ 3720 "subir" "breakAfter"
        movel(subir, a=0.01, v=0.01)
        $ 3721 "bajada_broca≔pose_sub(bajada_broca, bajada)"
        global bajada_broca= pose_sub (bajada_broca, bajada)
        Loop_100 = Loop_100 + 1
      end
      $ 3722 "Direction: Base Z+"
      global move_thread_flag_3722=0
      thread move_thread_3722():
        enter_critical
        move_thread_flag_3722 = 1
        local towardsPos=calculate_point_to_move_towards(p[0.0,0.0,0.0,0.0,0.0,0.0], [0.0,0.0,1.0], 0.06)
        movel(towardsPos, a=0.035, v=0.03)
        move_thread_flag_3722 = 2
        exit_critical
      end
      move_thread_flag_3722 = 0
      move_thread_han_3722 = run move_thread_3722()
      while (True):
        sleep(1.0E-10)
        if (move_thread_flag_3722 > 1):
          join move_thread_han_3722
          $ 3723 "Until (distance)"
          break
        end
        sync()
      end
      $ 3724 "Set CO[1]=Apagar"
      set_configurable_digital_out(1, False)
      $ 3725 "barreno_actual≔barreno_actual+1"
      global barreno_actual=barreno_actual+1
    end
    $ 3728 "Popup: Linea3 con full Terminada!"
    popup("Linea3 con full Terminada!", "Mensaje", False, False, blocking=True)
    $ 3729 "Linea4"
    $ 3730 "Marcar_puntos"
    $ 3731 "MoveL"
    $ 3732 "Home3" "breakAfter"
    movel(Home3_p, a=0.5, v=0.1)
    $ 3733 "Linea4_A" "breakAfter"
    movel(Linea4_A_p, a=0.5, v=0.1)
    $ 3734 "Linea4_B" "breakAfter"
    movel(Linea4_B_p, a=0.5, v=0.1)
    $ 3735 "Linea4_C" "breakAfter"
    movel(Linea4_C_p, a=0.5, v=0.1)
    $ 3736 "Linea4_D" "breakAfter"
    movel(Linea4_D_p, a=0.5, v=0.1)
    $ 3737 "Linea4_E" "breakAfter"
    movel(Linea4_E_p, a=0.5, v=0.1)
    $ 3738 "Linea4_F" "breakAfter"
    movel(Linea4_F_p, a=0.5, v=0.1)
    $ 3739 "AB"
    $ 3740 "'desbaste_inicial'"
    # 'desbaste_inicial'
    $ 3741 "bajada_broca≔p[0,0,-0.024,0,0,0]"
    global bajada_broca=p[0,0,-0.024,0,0,0]
    $ 3742 "barrenos_menos1≔8"
    global barrenos_menos1=8
    $ 3743 "barreno_actual≔0"
    global barreno_actual=0
    $ 3744 "Loop barreno_actual≤barrenos_menos1"
    while (barreno_actual <= barrenos_menos1):
      $ 3745 "Perforacion"
      $ 3746 "MoveL"
      $ 3747 "internos≔interpolate_pose(Linea4_A, Linea4_B, barreno_actual/barrenos_menos1)"
      global internos= interpolate_pose (Linea4_A_p, Linea4_B_p, barreno_actual/barrenos_menos1)
      $ 3748 "internos" "breakAfter"
      movel(internos, a=0.5, v=0.1)
      $ 3749 "'desbaste_inicial'"
      # 'desbaste_inicial'
      $ 3750 "bajada_broca≔p[0,0,-0.024,0,0,0]"
      global bajada_broca=p[0,0,-0.024,0,0,0]
      $ 3751 "bajada≔p[0,0,0.024,0,0,0]"
      global bajada=p[0,0,0.024,0,0,0]
      $ 3752 "Direction: Base Z-"
      global move_thread_flag_3752=0
      thread move_thread_3752():
        enter_critical
        move_thread_flag_3752 = 1
        local towardsPos=calculate_point_to_move_towards(p[0.0,0.0,0.0,0.0,0.0,0.0], [0.0,0.0,-1.0], 0.076)
        movel(towardsPos, a=0.015, v=0.02)
        move_thread_flag_3752 = 2
        exit_critical
      end
      move_thread_flag_3752 = 0
      move_thread_han_3752 = run move_thread_3752()
      while (True):
        sleep(1.0E-10)
        if (move_thread_flag_3752 > 1):
          join move_thread_han_3752
          $ 3753 "Until (distance)"
          break
        end
        sync()
      end
      $ 3754 "Popup: punto contacto alanzdo"
      popup("punto contacto alanzdo", "Mensaje", False, False, blocking=True)
      $ 3755 "Direction: Base Z+"
      global move_thread_flag_3755=0
      thread move_thread_3755():
        enter_critical
        move_thread_flag_3755 = 1
        local towardsPos=calculate_point_to_move_towards(p[0.0,0.0,0.0,0.0,0.0,0.0], [0.0,0.0,1.0], 0.002)
        movel(towardsPos, a=0.005, v=0.003)
        move_thread_flag_3755 = 2
        exit_critical
      end
      move_thread_flag_3755 = 0
      move_thread_han_3755 = run move_thread_3755()
      while (True):
        sleep(1.0E-10)
        if (move_thread_flag_3755 > 1):
          join move_thread_han_3755
          $ 3756 "Until (distance)"
          break
        end
        sync()
      end
      $ 3757 "Wait: 0.3"
      sleep(0.3)
      $ 3758 "Set CO[1]=Encender"
      set_configurable_digital_out(1, True)
      $ 3759 "Wait: 0.3"
      sleep(0.3)
      $ 3760 "Loop 1 times"
      Loop_120 = 0
      while (Loop_120 < 1):
        $ 3761 "bajar≔pose_add(get_actual_tcp_pose(), bajada_broca)"
        global bajar= pose_add ( get_actual_tcp_pose (), bajada_broca)
        $ 3762 "bajar" "breakAfter"
        movel(bajar, a=0.005, v=0.001)
        $ 3763 "subir≔pose_sub(get_actual_tcp_pose(), bajada_broca)"
        global subir= pose_sub ( get_actual_tcp_pose (), bajada_broca)
        $ 3764 "subir" "breakAfter"
        movel(subir, a=0.01, v=0.01)
        $ 3765 "bajada_broca≔pose_sub(bajada_broca, bajada)"
        global bajada_broca= pose_sub (bajada_broca, bajada)
        Loop_120 = Loop_120 + 1
      end
      $ 3766 "Direction: Base Z+"
      global move_thread_flag_3766=0
      thread move_thread_3766():
        enter_critical
        move_thread_flag_3766 = 1
        local towardsPos=calculate_point_to_move_towards(p[0.0,0.0,0.0,0.0,0.0,0.0], [0.0,0.0,1.0], 0.06)
        movel(towardsPos, a=0.035, v=0.03)
        move_thread_flag_3766 = 2
        exit_critical
      end
      move_thread_flag_3766 = 0
      move_thread_han_3766 = run move_thread_3766()
      while (True):
        sleep(1.0E-10)
        if (move_thread_flag_3766 > 1):
          join move_thread_han_3766
          $ 3767 "Until (distance)"
          break
        end
        sync()
      end
      $ 3768 "Set CO[1]=Apagar"
      set_configurable_digital_out(1, False)
      $ 3769 "barreno_actual≔barreno_actual+1"
      global barreno_actual=barreno_actual+1
    end
    $ 3772 "CD"
    $ 3773 "'desbaste_inicial'"
    # 'desbaste_inicial'
    $ 3774 "bajada_broca≔p[0,0,-0.024,0,0,0]"
    global bajada_broca=p[0,0,-0.024,0,0,0]
    $ 3775 "barrenos_menos1≔8"
    global barrenos_menos1=8
    $ 3776 "barreno_actual≔0"
    global barreno_actual=0
    $ 3777 "Loop barreno_actual≤barrenos_menos1"
    while (barreno_actual <= barrenos_menos1):
      $ 3778 "Perforacion"
      $ 3779 "MoveL"
      $ 3780 "internos≔interpolate_pose(Linea4_C, Linea4_D, barreno_actual/barrenos_menos1)"
      global internos= interpolate_pose (Linea4_C_p, Linea4_D_p, barreno_actual/barrenos_menos1)
      $ 3781 "internos" "breakAfter"
      movel(internos, a=0.5, v=0.1)
      $ 3782 "'desbaste_inicial'"
      # 'desbaste_inicial'
      $ 3783 "bajada_broca≔p[0,0,-0.024,0,0,0]"
      global bajada_broca=p[0,0,-0.024,0,0,0]
      $ 3784 "bajada≔p[0,0,0.024,0,0,0]"
      global bajada=p[0,0,0.024,0,0,0]
      $ 3785 "Direction: Base Z-"
      global move_thread_flag_3785=0
      thread move_thread_3785():
        enter_critical
        move_thread_flag_3785 = 1
        local towardsPos=calculate_point_to_move_towards(p[0.0,0.0,0.0,0.0,0.0,0.0], [0.0,0.0,-1.0], 0.076)
        movel(towardsPos, a=0.015, v=0.02)
        move_thread_flag_3785 = 2
        exit_critical
      end
      move_thread_flag_3785 = 0
      move_thread_han_3785 = run move_thread_3785()
      while (True):
        sleep(1.0E-10)
        if (move_thread_flag_3785 > 1):
          join move_thread_han_3785
          $ 3786 "Until (distance)"
          break
        end
        sync()
      end
      $ 3787 "Popup: punto contacto alanzdo"
      popup("punto contacto alanzdo", "Mensaje", False, False, blocking=True)
      $ 3788 "Direction: Base Z+"
      global move_thread_flag_3788=0
      thread move_thread_3788():
        enter_critical
        move_thread_flag_3788 = 1
        local towardsPos=calculate_point_to_move_towards(p[0.0,0.0,0.0,0.0,0.0,0.0], [0.0,0.0,1.0], 0.002)
        movel(towardsPos, a=0.005, v=0.003)
        move_thread_flag_3788 = 2
        exit_critical
      end
      move_thread_flag_3788 = 0
      move_thread_han_3788 = run move_thread_3788()
      while (True):
        sleep(1.0E-10)
        if (move_thread_flag_3788 > 1):
          join move_thread_han_3788
          $ 3789 "Until (distance)"
          break
        end
        sync()
      end
      $ 3790 "Wait: 0.3"
      sleep(0.3)
      $ 3791 "Set CO[1]=Encender"
      set_configurable_digital_out(1, True)
      $ 3792 "Wait: 0.3"
      sleep(0.3)
      $ 3793 "Loop 1 times"
      Loop_123 = 0
      while (Loop_123 < 1):
        $ 3794 "bajar≔pose_add(get_actual_tcp_pose(), bajada_broca)"
        global bajar= pose_add ( get_actual_tcp_pose (), bajada_broca)
        $ 3795 "bajar" "breakAfter"
        movel(bajar, a=0.005, v=0.001)
        $ 3796 "subir≔pose_sub(get_actual_tcp_pose(), bajada_broca)"
        global subir= pose_sub ( get_actual_tcp_pose (), bajada_broca)
        $ 3797 "subir" "breakAfter"
        movel(subir, a=0.01, v=0.01)
        $ 3798 "bajada_broca≔pose_sub(bajada_broca, bajada)"
        global bajada_broca= pose_sub (bajada_broca, bajada)
        Loop_123 = Loop_123 + 1
      end
      $ 3799 "Direction: Base Z+"
      global move_thread_flag_3799=0
      thread move_thread_3799():
        enter_critical
        move_thread_flag_3799 = 1
        local towardsPos=calculate_point_to_move_towards(p[0.0,0.0,0.0,0.0,0.0,0.0], [0.0,0.0,1.0], 0.06)
        movel(towardsPos, a=0.035, v=0.03)
        move_thread_flag_3799 = 2
        exit_critical
      end
      move_thread_flag_3799 = 0
      move_thread_han_3799 = run move_thread_3799()
      while (True):
        sleep(1.0E-10)
        if (move_thread_flag_3799 > 1):
          join move_thread_han_3799
          $ 3800 "Until (distance)"
          break
        end
        sync()
      end
      $ 3801 "Set CO[1]=Apagar"
      set_configurable_digital_out(1, False)
      $ 3802 "barreno_actual≔barreno_actual+1"
      global barreno_actual=barreno_actual+1
    end
    $ 3805 "EF"
    $ 3806 "'desbaste_inicial'"
    # 'desbaste_inicial'
    $ 3807 "bajada_broca≔p[0,0,-0.024,0,0,0]"
    global bajada_broca=p[0,0,-0.024,0,0,0]
    $ 3808 "barrenos_menos1≔8"
    global barrenos_menos1=8
    $ 3809 "barreno_actual≔0"
    global barreno_actual=0
    $ 3810 "Loop barreno_actual≤barrenos_menos1"
    while (barreno_actual <= barrenos_menos1):
      $ 3811 "Perforacion"
      $ 3812 "MoveL"
      $ 3813 "internos≔interpolate_pose(Linea4_E, Linea4_F, barreno_actual/barrenos_menos1)"
      global internos= interpolate_pose (Linea4_E_p, Linea4_F_p, barreno_actual/barrenos_menos1)
      $ 3814 "internos" "breakAfter"
      movel(internos, a=0.5, v=0.1)
      $ 3815 "'desbaste_inicial'"
      # 'desbaste_inicial'
      $ 3816 "bajada_broca≔p[0,0,-0.024,0,0,0]"
      global bajada_broca=p[0,0,-0.024,0,0,0]
      $ 3817 "bajada≔p[0,0,0.024,0,0,0]"
      global bajada=p[0,0,0.024,0,0,0]
      $ 3818 "Direction: Base Z-"
      global move_thread_flag_3818=0
      thread move_thread_3818():
        enter_critical
        move_thread_flag_3818 = 1
        local towardsPos=calculate_point_to_move_towards(p[0.0,0.0,0.0,0.0,0.0,0.0], [0.0,0.0,-1.0], 0.076)
        movel(towardsPos, a=0.015, v=0.02)
        move_thread_flag_3818 = 2
        exit_critical
      end
      move_thread_flag_3818 = 0
      move_thread_han_3818 = run move_thread_3818()
      while (True):
        sleep(1.0E-10)
        if (move_thread_flag_3818 > 1):
          join move_thread_han_3818
          $ 3819 "Until (distance)"
          break
        end
        sync()
      end
      $ 3820 "Popup: punto contacto alanzdo"
      popup("punto contacto alanzdo", "Mensaje", False, False, blocking=True)
      $ 3821 "Direction: Base Z+"
      global move_thread_flag_3821=0
      thread move_thread_3821():
        enter_critical
        move_thread_flag_3821 = 1
        local towardsPos=calculate_point_to_move_towards(p[0.0,0.0,0.0,0.0,0.0,0.0], [0.0,0.0,1.0], 0.002)
        movel(towardsPos, a=0.005, v=0.003)
        move_thread_flag_3821 = 2
        exit_critical
      end
      move_thread_flag_3821 = 0
      move_thread_han_3821 = run move_thread_3821()
      while (True):
        sleep(1.0E-10)
        if (move_thread_flag_3821 > 1):
          join move_thread_han_3821
          $ 3822 "Until (distance)"
          break
        end
        sync()
      end
      $ 3823 "Wait: 0.3"
      sleep(0.3)
      $ 3824 "Set CO[1]=Encender"
      set_configurable_digital_out(1, True)
      $ 3825 "Wait: 0.3"
      sleep(0.3)
      $ 3826 "Loop 1 times"
      Loop_125 = 0
      while (Loop_125 < 1):
        $ 3827 "bajar≔pose_add(get_actual_tcp_pose(), bajada_broca)"
        global bajar= pose_add ( get_actual_tcp_pose (), bajada_broca)
        $ 3828 "bajar" "breakAfter"
        movel(bajar, a=0.005, v=0.001)
        $ 3829 "subir≔pose_sub(get_actual_tcp_pose(), bajada_broca)"
        global subir= pose_sub ( get_actual_tcp_pose (), bajada_broca)
        $ 3830 "subir" "breakAfter"
        movel(subir, a=0.01, v=0.01)
        $ 3831 "bajada_broca≔pose_sub(bajada_broca, bajada)"
        global bajada_broca= pose_sub (bajada_broca, bajada)
        Loop_125 = Loop_125 + 1
      end
      $ 3832 "Direction: Base Z+"
      global move_thread_flag_3832=0
      thread move_thread_3832():
        enter_critical
        move_thread_flag_3832 = 1
        local towardsPos=calculate_point_to_move_towards(p[0.0,0.0,0.0,0.0,0.0,0.0], [0.0,0.0,1.0], 0.06)
        movel(towardsPos, a=0.035, v=0.03)
        move_thread_flag_3832 = 2
        exit_critical
      end
      move_thread_flag_3832 = 0
      move_thread_han_3832 = run move_thread_3832()
      while (True):
        sleep(1.0E-10)
        if (move_thread_flag_3832 > 1):
          join move_thread_han_3832
          $ 3833 "Until (distance)"
          break
        end
        sync()
      end
      $ 3834 "Set CO[1]=Apagar"
      set_configurable_digital_out(1, False)
      $ 3835 "barreno_actual≔barreno_actual+1"
      global barreno_actual=barreno_actual+1
      $ 3836 "If barreno_actual≥barrenos_menos1"
      if (barreno_actual >= barrenos_menos1):
        $ 3837 "cambiar_broca≔ True "
        global cambiar_broca=  True
      end
    end
    $ 3840 "Popup: Linea4 con full Terminada!"
    popup("Linea4 con full Terminada!", "Mensaje", False, False, blocking=True)
    $ 4061 "720"
    $ 4062 "Broca_1"
    $ 4063 "Linea19"
    $ 4064 "Marcar_puntos"
    $ 4065 "MoveL"
    $ 4066 "Home3" "breakAfter"
    movel(Home3_p, a=0.5, v=0.1)
    $ 4067 "Linea19_A" "breakAfter"
    movel(Linea19_A_p, a=0.5, v=0.1)
    $ 4068 "bajada_comprobacion"
    $ 4069 "Direction: Base Z-"
    global move_thread_flag_4069=0
    thread move_thread_4069():
      enter_critical
      move_thread_flag_4069 = 1
      local towardsPos=calculate_point_to_move_towards(p[0.0,0.0,0.0,0.0,0.0,0.0], [0.0,0.0,-1.0], 0.071)
      movel(towardsPos, a=0.15, v=0.1)
      move_thread_flag_4069 = 2
      exit_critical
    end
    move_thread_flag_4069 = 0
    move_thread_han_4069 = run move_thread_4069()
    while (True):
      sleep(1.0E-10)
      if (move_thread_flag_4069 > 1):
        join move_thread_han_4069
        $ 4070 "Until (distance)"
        break
      end
      sync()
    end
    $ 4071 "Direction: Base Z-"
    global move_thread_flag_4071=0
    thread move_thread_4071():
      enter_critical
      move_thread_flag_4071 = 1
      local towardsPos=calculate_point_to_move_towards(p[0.0,0.0,0.0,0.0,0.0,0.0], [0.0,0.0,-1.0], 1000.0)
      movel(towardsPos, a=0.007, v=0.007)
      move_thread_flag_4071 = 2
      exit_critical
    end
    move_thread_flag_4071 = 0
    move_thread_han_4071 = run move_thread_4071()
    while (True):
      local targetTcpDirection=get_target_tcp_speed()
      local stepsToRetract=tool_contact(direction=targetTcpDirection)
      if (stepsToRetract > 0):
        kill move_thread_han_4071
        stopl(0.02)
        local backTrackMovement=get_actual_joint_positions_history(stepsToRetract)
        local contactPose=get_forward_kin(backTrackMovement)
        local posDir=[targetTcpDirection[0],targetTcpDirection[1],targetTcpDirection[2]]
        local retractTo=contactPose
        if (norm(posDir) > 1e-6):
          local normalizedPosDir=normalize(posDir)
          local additionalRetraction=p[normalizedPosDir[0] * 0.0, normalizedPosDir[1] * 0.0, normalizedPosDir[2] * 0.0, 0, 0, 0]
          retractTo = pose_sub(contactPose, additionalRetraction)
        end
        movel(retractTo, a=0.02, v=0.1)
        $ 4072 "Until (tool_contact_detection)"
        break
      end
      sync()
    end
    $ 4073 "Direction: Base Z+"
    global move_thread_flag_4073=0
    thread move_thread_4073():
      enter_critical
      move_thread_flag_4073 = 1
      local towardsPos=calculate_point_to_move_towards(p[0.0,0.0,0.0,0.0,0.0,0.0], [0.0,0.0,1.0], 0.08)
      movel(towardsPos, a=0.15, v=0.1)
      move_thread_flag_4073 = 2
      exit_critical
    end
    move_thread_flag_4073 = 0
    move_thread_han_4073 = run move_thread_4073()
    while (True):
      sleep(1.0E-10)
      if (move_thread_flag_4073 > 1):
        join move_thread_han_4073
        $ 4074 "Until (distance)"
        break
      end
      sync()
    end
    $ 4075 "Linea19_B" "breakAfter"
    movel(Linea19_B_p, a=0.5, v=0.1)
    $ 4076 "bajada_comprobacion"
    $ 4077 "Direction: Base Z-"
    global move_thread_flag_4077=0
    thread move_thread_4077():
      enter_critical
      move_thread_flag_4077 = 1
      local towardsPos=calculate_point_to_move_towards(p[0.0,0.0,0.0,0.0,0.0,0.0], [0.0,0.0,-1.0], 0.071)
      movel(towardsPos, a=0.15, v=0.1)
      move_thread_flag_4077 = 2
      exit_critical
    end
    move_thread_flag_4077 = 0
    move_thread_han_4077 = run move_thread_4077()
    while (True):
      sleep(1.0E-10)
      if (move_thread_flag_4077 > 1):
        join move_thread_han_4077
        $ 4078 "Until (distance)"
        break
      end
      sync()
    end
    $ 4079 "Direction: Base Z-"
    global move_thread_flag_4079=0
    thread move_thread_4079():
      enter_critical
      move_thread_flag_4079 = 1
      local towardsPos=calculate_point_to_move_towards(p[0.0,0.0,0.0,0.0,0.0,0.0], [0.0,0.0,-1.0], 1000.0)
      movel(towardsPos, a=0.007, v=0.007)
      move_thread_flag_4079 = 2
      exit_critical
    end
    move_thread_flag_4079 = 0
    move_thread_han_4079 = run move_thread_4079()
    while (True):
      local targetTcpDirection=get_target_tcp_speed()
      local stepsToRetract=tool_contact(direction=targetTcpDirection)
      if (stepsToRetract > 0):
        kill move_thread_han_4079
        stopl(0.02)
        local backTrackMovement=get_actual_joint_positions_history(stepsToRetract)
        local contactPose=get_forward_kin(backTrackMovement)
        local posDir=[targetTcpDirection[0],targetTcpDirection[1],targetTcpDirection[2]]
        local retractTo=contactPose
        if (norm(posDir) > 1e-6):
          local normalizedPosDir=normalize(posDir)
          local additionalRetraction=p[normalizedPosDir[0] * 0.0, normalizedPosDir[1] * 0.0, normalizedPosDir[2] * 0.0, 0, 0, 0]
          retractTo = pose_sub(contactPose, additionalRetraction)
        end
        movel(retractTo, a=0.02, v=0.1)
        $ 4080 "Until (tool_contact_detection)"
        break
      end
      sync()
    end
    $ 4081 "Direction: Base Z+"
    global move_thread_flag_4081=0
    thread move_thread_4081():
      enter_critical
      move_thread_flag_4081 = 1
      local towardsPos=calculate_point_to_move_towards(p[0.0,0.0,0.0,0.0,0.0,0.0], [0.0,0.0,1.0], 0.08)
      movel(towardsPos, a=0.15, v=0.1)
      move_thread_flag_4081 = 2
      exit_critical
    end
    move_thread_flag_4081 = 0
    move_thread_han_4081 = run move_thread_4081()
    while (True):
      sleep(1.0E-10)
      if (move_thread_flag_4081 > 1):
        join move_thread_han_4081
        $ 4082 "Until (distance)"
        break
      end
      sync()
    end
    $ 4083 "AB"
    $ 4084 "'desbaste_inicial'"
    # 'desbaste_inicial'
    $ 4085 "bajada_broca≔p[0,0,-0.008,0,0,0]"
    global bajada_broca=p[0,0,-0.008,0,0,0]
    $ 4086 "barrenos_menos1≔1"
    global barrenos_menos1=1
    $ 4087 "barreno_actual≔0"
    global barreno_actual=0
    $ 4088 "Loop barreno_actual≤barrenos_menos1"
    while (barreno_actual <= barrenos_menos1):
      $ 4089 "Perforacion"
      $ 4090 "MoveL"
      $ 4091 "internos≔interpolate_pose(Linea19_A, Linea19_B, barreno_actual/barrenos_menos1)"
      global internos= interpolate_pose (Linea19_A_p, Linea19_B_p, barreno_actual/barrenos_menos1)
      $ 4092 "internos" "breakAfter"
      movel(internos, a=0.5, v=0.1)
      $ 4093 "'desbaste_inicial'"
      # 'desbaste_inicial'
      $ 4094 "bajada_broca≔p[0,0,-0.024,0,0,0]"
      global bajada_broca=p[0,0,-0.024,0,0,0]
      $ 4095 "bajada≔p[0,0,0.024,0,0,0]"
      global bajada=p[0,0,0.024,0,0,0]
      $ 4096 "Direction: Base Z-"
      global move_thread_flag_4096=0
      thread move_thread_4096():
        enter_critical
        move_thread_flag_4096 = 1
        local towardsPos=calculate_point_to_move_towards(p[0.0,0.0,0.0,0.0,0.0,0.0], [0.0,0.0,-1.0], 0.071)
        movel(towardsPos, a=0.15, v=0.1)
        move_thread_flag_4096 = 2
        exit_critical
      end
      move_thread_flag_4096 = 0
      move_thread_han_4096 = run move_thread_4096()
      while (True):
        sleep(1.0E-10)
        if (move_thread_flag_4096 > 1):
          join move_thread_han_4096
          $ 4097 "Until (distance)"
          break
        end
        sync()
      end
      $ 4098 "Direction: Base Z-"
      global move_thread_flag_4098=0
      thread move_thread_4098():
        enter_critical
        move_thread_flag_4098 = 1
        local towardsPos=calculate_point_to_move_towards(p[0.0,0.0,0.0,0.0,0.0,0.0], [0.0,0.0,-1.0], 1000.0)
        movel(towardsPos, a=0.007, v=0.007)
        move_thread_flag_4098 = 2
        exit_critical
      end
      move_thread_flag_4098 = 0
      move_thread_han_4098 = run move_thread_4098()
      while (True):
        local targetTcpDirection=get_target_tcp_speed()
        local stepsToRetract=tool_contact(direction=targetTcpDirection)
        if (stepsToRetract > 0):
          kill move_thread_han_4098
          stopl(0.02)
          local backTrackMovement=get_actual_joint_positions_history(stepsToRetract)
          local contactPose=get_forward_kin(backTrackMovement)
          local posDir=[targetTcpDirection[0],targetTcpDirection[1],targetTcpDirection[2]]
          local retractTo=contactPose
          if (norm(posDir) > 1e-6):
            local normalizedPosDir=normalize(posDir)
            local additionalRetraction=p[normalizedPosDir[0] * 0.0, normalizedPosDir[1] * 0.0, normalizedPosDir[2] * 0.0, 0, 0, 0]
            retractTo = pose_sub(contactPose, additionalRetraction)
          end
          movel(retractTo, a=0.02, v=0.1)
          $ 4099 "Until (tool_contact_detection)"
          break
        end
        sync()
      end
      $ 4100 "Popup: punto contacto alanzdo"
      popup("punto contacto alanzdo", "Mensaje", False, False, blocking=True)
      $ 4101 "Direction: Base Z+"
      global move_thread_flag_4101=0
      thread move_thread_4101():
        enter_critical
        move_thread_flag_4101 = 1
        local towardsPos=calculate_point_to_move_towards(p[0.0,0.0,0.0,0.0,0.0,0.0], [0.0,0.0,1.0], 0.007)
        movel(towardsPos, a=0.015, v=0.015)
        move_thread_flag_4101 = 2
        exit_critical
      end
      move_thread_flag_4101 = 0
      move_thread_han_4101 = run move_thread_4101()
      while (True):
        sleep(1.0E-10)
        if (move_thread_flag_4101 > 1):
          join move_thread_han_4101
          $ 4102 "Until (distance)"
          break
        end
        sync()
      end
      $ 4103 "Wait: 0.3"
      sleep(0.3)
      $ 4104 "Set CO[1]=Encender"
      set_configurable_digital_out(1, True)
      $ 4105 "Wait: 0.3"
      sleep(0.3)
      $ 4106 "Loop 1 times"
      Loop_47 = 0
      while (Loop_47 < 1):
        $ 4107 "bajar≔pose_add(get_actual_tcp_pose(), bajada_broca)"
        global bajar= pose_add ( get_actual_tcp_pose (), bajada_broca)
        $ 4108 "bajar" "breakAfter"
        movel(bajar, a=0.004, v=0.004)
        $ 4109 "subir≔pose_sub(get_actual_tcp_pose(), bajada_broca)"
        global subir= pose_sub ( get_actual_tcp_pose (), bajada_broca)
        $ 4110 "Direction: Base Z+"
        global move_thread_flag_4110=0
        thread move_thread_4110():
          enter_critical
          move_thread_flag_4110 = 1
          local towardsPos=calculate_point_to_move_towards(p[0.0,0.0,0.0,0.0,0.0,0.0], [0.0,0.0,1.0], 0.002)
          movel(towardsPos, a=0.015, v=0.015)
          move_thread_flag_4110 = 2
          exit_critical
        end
        move_thread_flag_4110 = 0
        move_thread_han_4110 = run move_thread_4110()
        while (True):
          sleep(1.0E-10)
          if (move_thread_flag_4110 > 1):
            join move_thread_han_4110
            $ 4111 "Until (distance)"
            break
          end
          sync()
        end
        $ 4112 "Set CO[1]=Apagar"
        set_configurable_digital_out(1, False)
        $ 4113 "subir" "breakAfter"
        movel(subir, a=0.015, v=0.015)
        $ 4114 "bajada_broca≔pose_sub(bajada_broca, bajada)"
        global bajada_broca= pose_sub (bajada_broca, bajada)
        Loop_47 = Loop_47 + 1
      end
      $ 4115 "Direction: Base Z+"
      global move_thread_flag_4115=0
      thread move_thread_4115():
        enter_critical
        move_thread_flag_4115 = 1
        local towardsPos=calculate_point_to_move_towards(p[0.0,0.0,0.0,0.0,0.0,0.0], [0.0,0.0,1.0], 0.08)
        movel(towardsPos, a=0.15, v=0.1)
        move_thread_flag_4115 = 2
        exit_critical
      end
      move_thread_flag_4115 = 0
      move_thread_han_4115 = run move_thread_4115()
      while (True):
        sleep(1.0E-10)
        if (move_thread_flag_4115 > 1):
          join move_thread_han_4115
          $ 4116 "Until (distance)"
          break
        end
        sync()
      end
      $ 4117 "Set CO[1]=Apagar"
      set_configurable_digital_out(1, False)
      $ 4118 "barreno_actual≔barreno_actual+1"
      global barreno_actual=barreno_actual+1
    end
    $ 4121 "Popup: Linea19 con chica Terminada!"
    popup("Linea19 con chica Terminada!", "Mensaje", False, False, blocking=True)
    $ 4122 "Linea20"
    $ 4123 "Marcar_puntos"
    $ 4124 "MoveL"
    $ 4125 "Linea20_A" "breakAfter"
    movel(Linea20_A_p, a=0.5, v=0.1)
    $ 4126 "bajada_comprobacion"
    $ 4127 "Direction: Base Z-"
    global move_thread_flag_4127=0
    thread move_thread_4127():
      enter_critical
      move_thread_flag_4127 = 1
      local towardsPos=calculate_point_to_move_towards(p[0.0,0.0,0.0,0.0,0.0,0.0], [0.0,0.0,-1.0], 0.071)
      movel(towardsPos, a=0.15, v=0.1)
      move_thread_flag_4127 = 2
      exit_critical
    end
    move_thread_flag_4127 = 0
    move_thread_han_4127 = run move_thread_4127()
    while (True):
      sleep(1.0E-10)
      if (move_thread_flag_4127 > 1):
        join move_thread_han_4127
        $ 4128 "Until (distance)"
        break
      end
      sync()
    end
    $ 4129 "Direction: Base Z-"
    global move_thread_flag_4129=0
    thread move_thread_4129():
      enter_critical
      move_thread_flag_4129 = 1
      local towardsPos=calculate_point_to_move_towards(p[0.0,0.0,0.0,0.0,0.0,0.0], [0.0,0.0,-1.0], 1000.0)
      movel(towardsPos, a=0.007, v=0.007)
      move_thread_flag_4129 = 2
      exit_critical
    end
    move_thread_flag_4129 = 0
    move_thread_han_4129 = run move_thread_4129()
    while (True):
      local targetTcpDirection=get_target_tcp_speed()
      local stepsToRetract=tool_contact(direction=targetTcpDirection)
      if (stepsToRetract > 0):
        kill move_thread_han_4129
        stopl(0.02)
        local backTrackMovement=get_actual_joint_positions_history(stepsToRetract)
        local contactPose=get_forward_kin(backTrackMovement)
        local posDir=[targetTcpDirection[0],targetTcpDirection[1],targetTcpDirection[2]]
        local retractTo=contactPose
        if (norm(posDir) > 1e-6):
          local normalizedPosDir=normalize(posDir)
          local additionalRetraction=p[normalizedPosDir[0] * 0.0, normalizedPosDir[1] * 0.0, normalizedPosDir[2] * 0.0, 0, 0, 0]
          retractTo = pose_sub(contactPose, additionalRetraction)
        end
        movel(retractTo, a=0.02, v=0.1)
        $ 4130 "Until (tool_contact_detection)"
        break
      end
      sync()
    end
    $ 4131 "Direction: Base Z+"
    global move_thread_flag_4131=0
    thread move_thread_4131():
      enter_critical
      move_thread_flag_4131 = 1
      local towardsPos=calculate_point_to_move_towards(p[0.0,0.0,0.0,0.0,0.0,0.0], [0.0,0.0,1.0], 0.08)
      movel(towardsPos, a=0.15, v=0.1)
      move_thread_flag_4131 = 2
      exit_critical
    end
    move_thread_flag_4131 = 0
    move_thread_han_4131 = run move_thread_4131()
    while (True):
      sleep(1.0E-10)
      if (move_thread_flag_4131 > 1):
        join move_thread_han_4131
        $ 4132 "Until (distance)"
        break
      end
      sync()
    end
    $ 4133 "Linea20_B" "breakAfter"
    movel(Linea20_B_p, a=0.5, v=0.1)
    $ 4134 "bajada_comprobacion"
    $ 4135 "Direction: Base Z-"
    global move_thread_flag_4135=0
    thread move_thread_4135():
      enter_critical
      move_thread_flag_4135 = 1
      local towardsPos=calculate_point_to_move_towards(p[0.0,0.0,0.0,0.0,0.0,0.0], [0.0,0.0,-1.0], 0.071)
      movel(towardsPos, a=0.15, v=0.1)
      move_thread_flag_4135 = 2
      exit_critical
    end
    move_thread_flag_4135 = 0
    move_thread_han_4135 = run move_thread_4135()
    while (True):
      sleep(1.0E-10)
      if (move_thread_flag_4135 > 1):
        join move_thread_han_4135
        $ 4136 "Until (distance)"
        break
      end
      sync()
    end
    $ 4137 "Direction: Base Z-"
    global move_thread_flag_4137=0
    thread move_thread_4137():
      enter_critical
      move_thread_flag_4137 = 1
      local towardsPos=calculate_point_to_move_towards(p[0.0,0.0,0.0,0.0,0.0,0.0], [0.0,0.0,-1.0], 1000.0)
      movel(towardsPos, a=0.007, v=0.007)
      move_thread_flag_4137 = 2
      exit_critical
    end
    move_thread_flag_4137 = 0
    move_thread_han_4137 = run move_thread_4137()
    while (True):
      local targetTcpDirection=get_target_tcp_speed()
      local stepsToRetract=tool_contact(direction=targetTcpDirection)
      if (stepsToRetract > 0):
        kill move_thread_han_4137
        stopl(0.02)
        local backTrackMovement=get_actual_joint_positions_history(stepsToRetract)
        local contactPose=get_forward_kin(backTrackMovement)
        local posDir=[targetTcpDirection[0],targetTcpDirection[1],targetTcpDirection[2]]
        local retractTo=contactPose
        if (norm(posDir) > 1e-6):
          local normalizedPosDir=normalize(posDir)
          local additionalRetraction=p[normalizedPosDir[0] * 0.0, normalizedPosDir[1] * 0.0, normalizedPosDir[2] * 0.0, 0, 0, 0]
          retractTo = pose_sub(contactPose, additionalRetraction)
        end
        movel(retractTo, a=0.02, v=0.1)
        $ 4138 "Until (tool_contact_detection)"
        break
      end
      sync()
    end
    $ 4139 "Direction: Base Z+"
    global move_thread_flag_4139=0
    thread move_thread_4139():
      enter_critical
      move_thread_flag_4139 = 1
      local towardsPos=calculate_point_to_move_towards(p[0.0,0.0,0.0,0.0,0.0,0.0], [0.0,0.0,1.0], 0.08)
      movel(towardsPos, a=0.15, v=0.1)
      move_thread_flag_4139 = 2
      exit_critical
    end
    move_thread_flag_4139 = 0
    move_thread_han_4139 = run move_thread_4139()
    while (True):
      sleep(1.0E-10)
      if (move_thread_flag_4139 > 1):
        join move_thread_han_4139
        $ 4140 "Until (distance)"
        break
      end
      sync()
    end
    $ 4141 "AB"
    $ 4142 "'desbaste_inicial'"
    # 'desbaste_inicial'
    $ 4143 "bajada_broca≔p[0,0,-0.008,0,0,0]"
    global bajada_broca=p[0,0,-0.008,0,0,0]
    $ 4144 "barrenos_menos1≔2"
    global barrenos_menos1=2
    $ 4145 "barreno_actual≔0"
    global barreno_actual=0
    $ 4146 "Loop barreno_actual≤barrenos_menos1"
    while (barreno_actual <= barrenos_menos1):
      $ 4147 "Perforacion"
      $ 4148 "MoveL"
      $ 4149 "internos≔interpolate_pose(Linea20_A, Linea20_B, barreno_actual/barrenos_menos1)"
      global internos= interpolate_pose (Linea20_A_p, Linea20_B_p, barreno_actual/barrenos_menos1)
      $ 4150 "internos" "breakAfter"
      movel(internos, a=0.5, v=0.1)
      $ 4151 "'desbaste_inicial'"
      # 'desbaste_inicial'
      $ 4152 "bajada_broca≔p[0,0,-0.024,0,0,0]"
      global bajada_broca=p[0,0,-0.024,0,0,0]
      $ 4153 "bajada≔p[0,0,0.024,0,0,0]"
      global bajada=p[0,0,0.024,0,0,0]
      $ 4154 "Direction: Base Z-"
      global move_thread_flag_4154=0
      thread move_thread_4154():
        enter_critical
        move_thread_flag_4154 = 1
        local towardsPos=calculate_point_to_move_towards(p[0.0,0.0,0.0,0.0,0.0,0.0], [0.0,0.0,-1.0], 0.071)
        movel(towardsPos, a=0.15, v=0.1)
        move_thread_flag_4154 = 2
        exit_critical
      end
      move_thread_flag_4154 = 0
      move_thread_han_4154 = run move_thread_4154()
      while (True):
        sleep(1.0E-10)
        if (move_thread_flag_4154 > 1):
          join move_thread_han_4154
          $ 4155 "Until (distance)"
          break
        end
        sync()
      end
      $ 4156 "Direction: Base Z-"
      global move_thread_flag_4156=0
      thread move_thread_4156():
        enter_critical
        move_thread_flag_4156 = 1
        local towardsPos=calculate_point_to_move_towards(p[0.0,0.0,0.0,0.0,0.0,0.0], [0.0,0.0,-1.0], 1000.0)
        movel(towardsPos, a=0.007, v=0.007)
        move_thread_flag_4156 = 2
        exit_critical
      end
      move_thread_flag_4156 = 0
      move_thread_han_4156 = run move_thread_4156()
      while (True):
        local targetTcpDirection=get_target_tcp_speed()
        local stepsToRetract=tool_contact(direction=targetTcpDirection)
        if (stepsToRetract > 0):
          kill move_thread_han_4156
          stopl(0.02)
          local backTrackMovement=get_actual_joint_positions_history(stepsToRetract)
          local contactPose=get_forward_kin(backTrackMovement)
          local posDir=[targetTcpDirection[0],targetTcpDirection[1],targetTcpDirection[2]]
          local retractTo=contactPose
          if (norm(posDir) > 1e-6):
            local normalizedPosDir=normalize(posDir)
            local additionalRetraction=p[normalizedPosDir[0] * 0.0, normalizedPosDir[1] * 0.0, normalizedPosDir[2] * 0.0, 0, 0, 0]
            retractTo = pose_sub(contactPose, additionalRetraction)
          end
          movel(retractTo, a=0.02, v=0.1)
          $ 4157 "Until (tool_contact_detection)"
          break
        end
        sync()
      end
      $ 4158 "Popup: punto contacto alanzdo"
      popup("punto contacto alanzdo", "Mensaje", False, False, blocking=True)
      $ 4159 "Direction: Base Z+"
      global move_thread_flag_4159=0
      thread move_thread_4159():
        enter_critical
        move_thread_flag_4159 = 1
        local towardsPos=calculate_point_to_move_towards(p[0.0,0.0,0.0,0.0,0.0,0.0], [0.0,0.0,1.0], 0.007)
        movel(towardsPos, a=0.015, v=0.015)
        move_thread_flag_4159 = 2
        exit_critical
      end
      move_thread_flag_4159 = 0
      move_thread_han_4159 = run move_thread_4159()
      while (True):
        sleep(1.0E-10)
        if (move_thread_flag_4159 > 1):
          join move_thread_han_4159
          $ 4160 "Until (distance)"
          break
        end
        sync()
      end
      $ 4161 "Wait: 0.3"
      sleep(0.3)
      $ 4162 "Set CO[1]=Encender"
      set_configurable_digital_out(1, True)
      $ 4163 "Wait: 0.3"
      sleep(0.3)
      $ 4164 "Loop 1 times"
      Loop_57 = 0
      while (Loop_57 < 1):
        $ 4165 "bajar≔pose_add(get_actual_tcp_pose(), bajada_broca)"
        global bajar= pose_add ( get_actual_tcp_pose (), bajada_broca)
        $ 4166 "bajar" "breakAfter"
        movel(bajar, a=0.004, v=0.004)
        $ 4167 "subir≔pose_sub(get_actual_tcp_pose(), bajada_broca)"
        global subir= pose_sub ( get_actual_tcp_pose (), bajada_broca)
        $ 4168 "Direction: Base Z+"
        global move_thread_flag_4168=0
        thread move_thread_4168():
          enter_critical
          move_thread_flag_4168 = 1
          local towardsPos=calculate_point_to_move_towards(p[0.0,0.0,0.0,0.0,0.0,0.0], [0.0,0.0,1.0], 0.002)
          movel(towardsPos, a=0.015, v=0.015)
          move_thread_flag_4168 = 2
          exit_critical
        end
        move_thread_flag_4168 = 0
        move_thread_han_4168 = run move_thread_4168()
        while (True):
          sleep(1.0E-10)
          if (move_thread_flag_4168 > 1):
            join move_thread_han_4168
            $ 4169 "Until (distance)"
            break
          end
          sync()
        end
        $ 4170 "Set CO[1]=Apagar"
        set_configurable_digital_out(1, False)
        $ 4171 "subir" "breakAfter"
        movel(subir, a=0.015, v=0.015)
        $ 4172 "bajada_broca≔pose_sub(bajada_broca, bajada)"
        global bajada_broca= pose_sub (bajada_broca, bajada)
        Loop_57 = Loop_57 + 1
      end
      $ 4173 "Direction: Base Z+"
      global move_thread_flag_4173=0
      thread move_thread_4173():
        enter_critical
        move_thread_flag_4173 = 1
        local towardsPos=calculate_point_to_move_towards(p[0.0,0.0,0.0,0.0,0.0,0.0], [0.0,0.0,1.0], 0.08)
        movel(towardsPos, a=0.15, v=0.1)
        move_thread_flag_4173 = 2
        exit_critical
      end
      move_thread_flag_4173 = 0
      move_thread_han_4173 = run move_thread_4173()
      while (True):
        sleep(1.0E-10)
        if (move_thread_flag_4173 > 1):
          join move_thread_han_4173
          $ 4174 "Until (distance)"
          break
        end
        sync()
      end
      $ 4175 "Set CO[1]=Apagar"
      set_configurable_digital_out(1, False)
      $ 4176 "barreno_actual≔barreno_actual+1"
      global barreno_actual=barreno_actual+1
    end
    $ 4179 "Popup: Linea20 con chica Terminada!"
    popup("Linea20 con chica Terminada!", "Mensaje", False, False, blocking=True)
    $ 4303 "Linea22"
    $ 4304 "Marcar_puntos"
    $ 4305 "MoveL"
    $ 4306 "Linea22_A" "breakAfter"
    movel(Linea22_A_p, a=0.5, v=0.1)
    $ 4307 "bajada_comprobacion"
    $ 4308 "Direction: Base Z-"
    global move_thread_flag_4308=0
    thread move_thread_4308():
      enter_critical
      move_thread_flag_4308 = 1
      local towardsPos=calculate_point_to_move_towards(p[0.0,0.0,0.0,0.0,0.0,0.0], [0.0,0.0,-1.0], 0.071)
      movel(towardsPos, a=0.15, v=0.1)
      move_thread_flag_4308 = 2
      exit_critical
    end
    move_thread_flag_4308 = 0
    move_thread_han_4308 = run move_thread_4308()
    while (True):
      sleep(1.0E-10)
      if (move_thread_flag_4308 > 1):
        join move_thread_han_4308
        $ 4309 "Until (distance)"
        break
      end
      sync()
    end
    $ 4310 "Direction: Base Z-"
    global move_thread_flag_4310=0
    thread move_thread_4310():
      enter_critical
      move_thread_flag_4310 = 1
      local towardsPos=calculate_point_to_move_towards(p[0.0,0.0,0.0,0.0,0.0,0.0], [0.0,0.0,-1.0], 1000.0)
      movel(towardsPos, a=0.007, v=0.007)
      move_thread_flag_4310 = 2
      exit_critical
    end
    move_thread_flag_4310 = 0
    move_thread_han_4310 = run move_thread_4310()
    while (True):
      local targetTcpDirection=get_target_tcp_speed()
      local stepsToRetract=tool_contact(direction=targetTcpDirection)
      if (stepsToRetract > 0):
        kill move_thread_han_4310
        stopl(0.02)
        local backTrackMovement=get_actual_joint_positions_history(stepsToRetract)
        local contactPose=get_forward_kin(backTrackMovement)
        local posDir=[targetTcpDirection[0],targetTcpDirection[1],targetTcpDirection[2]]
        local retractTo=contactPose
        if (norm(posDir) > 1e-6):
          local normalizedPosDir=normalize(posDir)
          local additionalRetraction=p[normalizedPosDir[0] * 0.0, normalizedPosDir[1] * 0.0, normalizedPosDir[2] * 0.0, 0, 0, 0]
          retractTo = pose_sub(contactPose, additionalRetraction)
        end
        movel(retractTo, a=0.02, v=0.1)
        $ 4311 "Until (tool_contact_detection)"
        break
      end
      sync()
    end
    $ 4312 "Direction: Base Z+"
    global move_thread_flag_4312=0
    thread move_thread_4312():
      enter_critical
      move_thread_flag_4312 = 1
      local towardsPos=calculate_point_to_move_towards(p[0.0,0.0,0.0,0.0,0.0,0.0], [0.0,0.0,1.0], 0.08)
      movel(towardsPos, a=0.15, v=0.1)
      move_thread_flag_4312 = 2
      exit_critical
    end
    move_thread_flag_4312 = 0
    move_thread_han_4312 = run move_thread_4312()
    while (True):
      sleep(1.0E-10)
      if (move_thread_flag_4312 > 1):
        join move_thread_han_4312
        $ 4313 "Until (distance)"
        break
      end
      sync()
    end
    $ 4314 "Linea22_B" "breakAfter"
    movel(Linea22_B_p, a=0.5, v=0.1)
    $ 4315 "bajada_comprobacion"
    $ 4316 "Direction: Base Z-"
    global move_thread_flag_4316=0
    thread move_thread_4316():
      enter_critical
      move_thread_flag_4316 = 1
      local towardsPos=calculate_point_to_move_towards(p[0.0,0.0,0.0,0.0,0.0,0.0], [0.0,0.0,-1.0], 0.071)
      movel(towardsPos, a=0.15, v=0.1)
      move_thread_flag_4316 = 2
      exit_critical
    end
    move_thread_flag_4316 = 0
    move_thread_han_4316 = run move_thread_4316()
    while (True):
      sleep(1.0E-10)
      if (move_thread_flag_4316 > 1):
        join move_thread_han_4316
        $ 4317 "Until (distance)"
        break
      end
      sync()
    end
    $ 4318 "Direction: Base Z-"
    global move_thread_flag_4318=0
    thread move_thread_4318():
      enter_critical
      move_thread_flag_4318 = 1
      local towardsPos=calculate_point_to_move_towards(p[0.0,0.0,0.0,0.0,0.0,0.0], [0.0,0.0,-1.0], 1000.0)
      movel(towardsPos, a=0.007, v=0.007)
      move_thread_flag_4318 = 2
      exit_critical
    end
    move_thread_flag_4318 = 0
    move_thread_han_4318 = run move_thread_4318()
    while (True):
      local targetTcpDirection=get_target_tcp_speed()
      local stepsToRetract=tool_contact(direction=targetTcpDirection)
      if (stepsToRetract > 0):
        kill move_thread_han_4318
        stopl(0.02)
        local backTrackMovement=get_actual_joint_positions_history(stepsToRetract)
        local contactPose=get_forward_kin(backTrackMovement)
        local posDir=[targetTcpDirection[0],targetTcpDirection[1],targetTcpDirection[2]]
        local retractTo=contactPose
        if (norm(posDir) > 1e-6):
          local normalizedPosDir=normalize(posDir)
          local additionalRetraction=p[normalizedPosDir[0] * 0.0, normalizedPosDir[1] * 0.0, normalizedPosDir[2] * 0.0, 0, 0, 0]
          retractTo = pose_sub(contactPose, additionalRetraction)
        end
        movel(retractTo, a=0.02, v=0.1)
        $ 4319 "Until (tool_contact_detection)"
        break
      end
      sync()
    end
    $ 4320 "Direction: Base Z+"
    global move_thread_flag_4320=0
    thread move_thread_4320():
      enter_critical
      move_thread_flag_4320 = 1
      local towardsPos=calculate_point_to_move_towards(p[0.0,0.0,0.0,0.0,0.0,0.0], [0.0,0.0,1.0], 0.08)
      movel(towardsPos, a=0.15, v=0.1)
      move_thread_flag_4320 = 2
      exit_critical
    end
    move_thread_flag_4320 = 0
    move_thread_han_4320 = run move_thread_4320()
    while (True):
      sleep(1.0E-10)
      if (move_thread_flag_4320 > 1):
        join move_thread_han_4320
        $ 4321 "Until (distance)"
        break
      end
      sync()
    end
    $ 4322 "AB"
    $ 4323 "'desbaste_inicial'"
    # 'desbaste_inicial'
    $ 4324 "bajada_broca≔p[0,0,-0.008,0,0,0]"
    global bajada_broca=p[0,0,-0.008,0,0,0]
    $ 4325 "barrenos_menos1≔1"
    global barrenos_menos1=1
    $ 4326 "barreno_actual≔0"
    global barreno_actual=0
    $ 4327 "Loop barreno_actual≤barrenos_menos1"
    while (barreno_actual <= barrenos_menos1):
      $ 4328 "Perforacion"
      $ 4329 "MoveL"
      $ 4332 "internos≔interpolate_pose(Linea22_A, Linea22_B, barreno_actual/barrenos_menos1)"
      global internos= interpolate_pose (Linea22_A_p, Linea22_B_p, barreno_actual/barrenos_menos1)
      $ 4333 "internos" "breakAfter"
      movel(internos, a=0.5, v=0.1)
      $ 4334 "'desbaste_inicial'"
      # 'desbaste_inicial'
      $ 4335 "bajada_broca≔p[0,0,-0.024,0,0,0]"
      global bajada_broca=p[0,0,-0.024,0,0,0]
      $ 4336 "bajada≔p[0,0,0.024,0,0,0]"
      global bajada=p[0,0,0.024,0,0,0]
      $ 4337 "Direction: Base Z-"
      global move_thread_flag_4337=0
      thread move_thread_4337():
        enter_critical
        move_thread_flag_4337 = 1
        local towardsPos=calculate_point_to_move_towards(p[0.0,0.0,0.0,0.0,0.0,0.0], [0.0,0.0,-1.0], 0.071)
        movel(towardsPos, a=0.15, v=0.1)
        move_thread_flag_4337 = 2
        exit_critical
      end
      move_thread_flag_4337 = 0
      move_thread_han_4337 = run move_thread_4337()
      while (True):
        sleep(1.0E-10)
        if (move_thread_flag_4337 > 1):
          join move_thread_han_4337
          $ 4338 "Until (distance)"
          break
        end
        sync()
      end
      $ 4339 "Direction: Base Z-"
      global move_thread_flag_4339=0
      thread move_thread_4339():
        enter_critical
        move_thread_flag_4339 = 1
        local towardsPos=calculate_point_to_move_towards(p[0.0,0.0,0.0,0.0,0.0,0.0], [0.0,0.0,-1.0], 1000.0)
        movel(towardsPos, a=0.007, v=0.007)
        move_thread_flag_4339 = 2
        exit_critical
      end
      move_thread_flag_4339 = 0
      move_thread_han_4339 = run move_thread_4339()
      while (True):
        local targetTcpDirection=get_target_tcp_speed()
        local stepsToRetract=tool_contact(direction=targetTcpDirection)
        if (stepsToRetract > 0):
          kill move_thread_han_4339
          stopl(0.02)
          local backTrackMovement=get_actual_joint_positions_history(stepsToRetract)
          local contactPose=get_forward_kin(backTrackMovement)
          local posDir=[targetTcpDirection[0],targetTcpDirection[1],targetTcpDirection[2]]
          local retractTo=contactPose
          if (norm(posDir) > 1e-6):
            local normalizedPosDir=normalize(posDir)
            local additionalRetraction=p[normalizedPosDir[0] * 0.0, normalizedPosDir[1] * 0.0, normalizedPosDir[2] * 0.0, 0, 0, 0]
            retractTo = pose_sub(contactPose, additionalRetraction)
          end
          movel(retractTo, a=0.02, v=0.1)
          $ 4340 "Until (tool_contact_detection)"
          break
        end
        sync()
      end
      $ 4341 "Popup: punto contacto alanzdo"
      popup("punto contacto alanzdo", "Mensaje", False, False, blocking=True)
      $ 4342 "Direction: Base Z+"
      global move_thread_flag_4342=0
      thread move_thread_4342():
        enter_critical
        move_thread_flag_4342 = 1
        local towardsPos=calculate_point_to_move_towards(p[0.0,0.0,0.0,0.0,0.0,0.0], [0.0,0.0,1.0], 0.007)
        movel(towardsPos, a=0.015, v=0.015)
        move_thread_flag_4342 = 2
        exit_critical
      end
      move_thread_flag_4342 = 0
      move_thread_han_4342 = run move_thread_4342()
      while (True):
        sleep(1.0E-10)
        if (move_thread_flag_4342 > 1):
          join move_thread_han_4342
          $ 4343 "Until (distance)"
          break
        end
        sync()
      end
      $ 4344 "Wait: 0.3"
      sleep(0.3)
      $ 4345 "Set CO[1]=Encender"
      set_configurable_digital_out(1, True)
      $ 4346 "Wait: 0.3"
      sleep(0.3)
      $ 4347 "Loop 1 times"
      Loop_84 = 0
      while (Loop_84 < 1):
        $ 4348 "bajar≔pose_add(get_actual_tcp_pose(), bajada_broca)"
        global bajar= pose_add ( get_actual_tcp_pose (), bajada_broca)
        $ 4349 "bajar" "breakAfter"
        movel(bajar, a=0.004, v=0.004)
        $ 4350 "subir≔pose_sub(get_actual_tcp_pose(), bajada_broca)"
        global subir= pose_sub ( get_actual_tcp_pose (), bajada_broca)
        $ 4351 "Direction: Base Z+"
        global move_thread_flag_4351=0
        thread move_thread_4351():
          enter_critical
          move_thread_flag_4351 = 1
          local towardsPos=calculate_point_to_move_towards(p[0.0,0.0,0.0,0.0,0.0,0.0], [0.0,0.0,1.0], 0.002)
          movel(towardsPos, a=0.015, v=0.015)
          move_thread_flag_4351 = 2
          exit_critical
        end
        move_thread_flag_4351 = 0
        move_thread_han_4351 = run move_thread_4351()
        while (True):
          sleep(1.0E-10)
          if (move_thread_flag_4351 > 1):
            join move_thread_han_4351
            $ 4352 "Until (distance)"
            break
          end
          sync()
        end
        $ 4353 "Set CO[1]=Apagar"
        set_configurable_digital_out(1, False)
        $ 4354 "subir" "breakAfter"
        movel(subir, a=0.01, v=0.005)
        $ 4355 "bajada_broca≔pose_sub(bajada_broca, bajada)"
        global bajada_broca= pose_sub (bajada_broca, bajada)
        Loop_84 = Loop_84 + 1
      end
      $ 4356 "Direction: Base Z+"
      global move_thread_flag_4356=0
      thread move_thread_4356():
        enter_critical
        move_thread_flag_4356 = 1
        local towardsPos=calculate_point_to_move_towards(p[0.0,0.0,0.0,0.0,0.0,0.0], [0.0,0.0,1.0], 0.08)
        movel(towardsPos, a=0.15, v=0.1)
        move_thread_flag_4356 = 2
        exit_critical
      end
      move_thread_flag_4356 = 0
      move_thread_han_4356 = run move_thread_4356()
      while (True):
        sleep(1.0E-10)
        if (move_thread_flag_4356 > 1):
          join move_thread_han_4356
          $ 4357 "Until (distance)"
          break
        end
        sync()
      end
      $ 4358 "Set CO[1]=Apagar"
      set_configurable_digital_out(1, False)
      $ 4359 "barreno_actual≔barreno_actual+1"
      global barreno_actual=barreno_actual+1
    end
    $ 4362 "Popup: Linea22 con chica Terminada!"
    popup("Linea22 con chica Terminada!", "Mensaje", False, False, blocking=True)
    $ 4363 "Linea23"
    $ 4364 "Marcar_puntos"
    $ 4365 "MoveL"
    $ 4366 "Linea23_A" "breakAfter"
    movel(Linea23_A_p, a=0.5, v=0.1)
    $ 4367 "bajada_comprobacion"
    $ 4368 "Direction: Base Z-"
    global move_thread_flag_4368=0
    thread move_thread_4368():
      enter_critical
      move_thread_flag_4368 = 1
      local towardsPos=calculate_point_to_move_towards(p[0.0,0.0,0.0,0.0,0.0,0.0], [0.0,0.0,-1.0], 0.071)
      movel(towardsPos, a=0.15, v=0.1)
      move_thread_flag_4368 = 2
      exit_critical
    end
    move_thread_flag_4368 = 0
    move_thread_han_4368 = run move_thread_4368()
    while (True):
      sleep(1.0E-10)
      if (move_thread_flag_4368 > 1):
        join move_thread_han_4368
        $ 4369 "Until (distance)"
        break
      end
      sync()
    end
    $ 4370 "Direction: Base Z-"
    global move_thread_flag_4370=0
    thread move_thread_4370():
      enter_critical
      move_thread_flag_4370 = 1
      local towardsPos=calculate_point_to_move_towards(p[0.0,0.0,0.0,0.0,0.0,0.0], [0.0,0.0,-1.0], 1000.0)
      movel(towardsPos, a=0.007, v=0.007)
      move_thread_flag_4370 = 2
      exit_critical
    end
    move_thread_flag_4370 = 0
    move_thread_han_4370 = run move_thread_4370()
    while (True):
      local targetTcpDirection=get_target_tcp_speed()
      local stepsToRetract=tool_contact(direction=targetTcpDirection)
      if (stepsToRetract > 0):
        kill move_thread_han_4370
        stopl(0.02)
        local backTrackMovement=get_actual_joint_positions_history(stepsToRetract)
        local contactPose=get_forward_kin(backTrackMovement)
        local posDir=[targetTcpDirection[0],targetTcpDirection[1],targetTcpDirection[2]]
        local retractTo=contactPose
        if (norm(posDir) > 1e-6):
          local normalizedPosDir=normalize(posDir)
          local additionalRetraction=p[normalizedPosDir[0] * 0.0, normalizedPosDir[1] * 0.0, normalizedPosDir[2] * 0.0, 0, 0, 0]
          retractTo = pose_sub(contactPose, additionalRetraction)
        end
        movel(retractTo, a=0.02, v=0.1)
        $ 4371 "Until (tool_contact_detection)"
        break
      end
      sync()
    end
    $ 4372 "Direction: Base Z+"
    global move_thread_flag_4372=0
    thread move_thread_4372():
      enter_critical
      move_thread_flag_4372 = 1
      local towardsPos=calculate_point_to_move_towards(p[0.0,0.0,0.0,0.0,0.0,0.0], [0.0,0.0,1.0], 0.08)
      movel(towardsPos, a=0.15, v=0.1)
      move_thread_flag_4372 = 2
      exit_critical
    end
    move_thread_flag_4372 = 0
    move_thread_han_4372 = run move_thread_4372()
    while (True):
      sleep(1.0E-10)
      if (move_thread_flag_4372 > 1):
        join move_thread_han_4372
        $ 4373 "Until (distance)"
        break
      end
      sync()
    end
    $ 4374 "Linea23_B" "breakAfter"
    movel(Linea23_B_p, a=0.5, v=0.1)
    $ 4375 "bajada_comprobacion"
    $ 4376 "Direction: Base Z-"
    global move_thread_flag_4376=0
    thread move_thread_4376():
      enter_critical
      move_thread_flag_4376 = 1
      local towardsPos=calculate_point_to_move_towards(p[0.0,0.0,0.0,0.0,0.0,0.0], [0.0,0.0,-1.0], 0.071)
      movel(towardsPos, a=0.15, v=0.1)
      move_thread_flag_4376 = 2
      exit_critical
    end
    move_thread_flag_4376 = 0
    move_thread_han_4376 = run move_thread_4376()
    while (True):
      sleep(1.0E-10)
      if (move_thread_flag_4376 > 1):
        join move_thread_han_4376
        $ 4377 "Until (distance)"
        break
      end
      sync()
    end
    $ 4378 "Direction: Base Z-"
    global move_thread_flag_4378=0
    thread move_thread_4378():
      enter_critical
      move_thread_flag_4378 = 1
      local towardsPos=calculate_point_to_move_towards(p[0.0,0.0,0.0,0.0,0.0,0.0], [0.0,0.0,-1.0], 1000.0)
      movel(towardsPos, a=0.007, v=0.007)
      move_thread_flag_4378 = 2
      exit_critical
    end
    move_thread_flag_4378 = 0
    move_thread_han_4378 = run move_thread_4378()
    while (True):
      local targetTcpDirection=get_target_tcp_speed()
      local stepsToRetract=tool_contact(direction=targetTcpDirection)
      if (stepsToRetract > 0):
        kill move_thread_han_4378
        stopl(0.02)
        local backTrackMovement=get_actual_joint_positions_history(stepsToRetract)
        local contactPose=get_forward_kin(backTrackMovement)
        local posDir=[targetTcpDirection[0],targetTcpDirection[1],targetTcpDirection[2]]
        local retractTo=contactPose
        if (norm(posDir) > 1e-6):
          local normalizedPosDir=normalize(posDir)
          local additionalRetraction=p[normalizedPosDir[0] * 0.0, normalizedPosDir[1] * 0.0, normalizedPosDir[2] * 0.0, 0, 0, 0]
          retractTo = pose_sub(contactPose, additionalRetraction)
        end
        movel(retractTo, a=0.02, v=0.1)
        $ 4379 "Until (tool_contact_detection)"
        break
      end
      sync()
    end
    $ 4380 "Direction: Base Z+"
    global move_thread_flag_4380=0
    thread move_thread_4380():
      enter_critical
      move_thread_flag_4380 = 1
      local towardsPos=calculate_point_to_move_towards(p[0.0,0.0,0.0,0.0,0.0,0.0], [0.0,0.0,1.0], 0.08)
      movel(towardsPos, a=0.15, v=0.1)
      move_thread_flag_4380 = 2
      exit_critical
    end
    move_thread_flag_4380 = 0
    move_thread_han_4380 = run move_thread_4380()
    while (True):
      sleep(1.0E-10)
      if (move_thread_flag_4380 > 1):
        join move_thread_han_4380
        $ 4381 "Until (distance)"
        break
      end
      sync()
    end
    $ 4382 "AB"
    $ 4383 "'desbaste_inicial'"
    # 'desbaste_inicial'
    $ 4384 "bajada_broca≔p[0,0,-0.008,0,0,0]"
    global bajada_broca=p[0,0,-0.008,0,0,0]
    $ 4385 "barrenos_menos1≔2"
    global barrenos_menos1=2
    $ 4386 "barreno_actual≔0"
    global barreno_actual=0
    $ 4387 "Loop barreno_actual≤barrenos_menos1"
    while (barreno_actual <= barrenos_menos1):
      $ 4388 "Perforacion"
      $ 4389 "MoveL"
      $ 4392 "internos≔interpolate_pose(Linea23_A, Linea23_B, barreno_actual/barrenos_menos1)"
      global internos= interpolate_pose (Linea23_A_p, Linea23_B_p, barreno_actual/barrenos_menos1)
      $ 4393 "internos" "breakAfter"
      movel(internos, a=0.5, v=0.1)
      $ 4394 "'desbaste_inicial'"
      # 'desbaste_inicial'
      $ 4395 "bajada_broca≔p[0,0,-0.024,0,0,0]"
      global bajada_broca=p[0,0,-0.024,0,0,0]
      $ 4396 "bajada≔p[0,0,0.024,0,0,0]"
      global bajada=p[0,0,0.024,0,0,0]
      $ 4397 "Direction: Base Z-"
      global move_thread_flag_4397=0
      thread move_thread_4397():
        enter_critical
        move_thread_flag_4397 = 1
        local towardsPos=calculate_point_to_move_towards(p[0.0,0.0,0.0,0.0,0.0,0.0], [0.0,0.0,-1.0], 0.071)
        movel(towardsPos, a=0.15, v=0.1)
        move_thread_flag_4397 = 2
        exit_critical
      end
      move_thread_flag_4397 = 0
      move_thread_han_4397 = run move_thread_4397()
      while (True):
        sleep(1.0E-10)
        if (move_thread_flag_4397 > 1):
          join move_thread_han_4397
          $ 4398 "Until (distance)"
          break
        end
        sync()
      end
      $ 4399 "Direction: Base Z-"
      global move_thread_flag_4399=0
      thread move_thread_4399():
        enter_critical
        move_thread_flag_4399 = 1
        local towardsPos=calculate_point_to_move_towards(p[0.0,0.0,0.0,0.0,0.0,0.0], [0.0,0.0,-1.0], 1000.0)
        movel(towardsPos, a=0.007, v=0.007)
        move_thread_flag_4399 = 2
        exit_critical
      end
      move_thread_flag_4399 = 0
      move_thread_han_4399 = run move_thread_4399()
      while (True):
        local targetTcpDirection=get_target_tcp_speed()
        local stepsToRetract=tool_contact(direction=targetTcpDirection)
        if (stepsToRetract > 0):
          kill move_thread_han_4399
          stopl(0.02)
          local backTrackMovement=get_actual_joint_positions_history(stepsToRetract)
          local contactPose=get_forward_kin(backTrackMovement)
          local posDir=[targetTcpDirection[0],targetTcpDirection[1],targetTcpDirection[2]]
          local retractTo=contactPose
          if (norm(posDir) > 1e-6):
            local normalizedPosDir=normalize(posDir)
            local additionalRetraction=p[normalizedPosDir[0] * 0.0, normalizedPosDir[1] * 0.0, normalizedPosDir[2] * 0.0, 0, 0, 0]
            retractTo = pose_sub(contactPose, additionalRetraction)
          end
          movel(retractTo, a=0.02, v=0.1)
          $ 4400 "Until (tool_contact_detection)"
          break
        end
        sync()
      end
      $ 4401 "Popup: punto contacto alanzdo"
      popup("punto contacto alanzdo", "Mensaje", False, False, blocking=True)
      $ 4402 "Direction: Base Z+"
      global move_thread_flag_4402=0
      thread move_thread_4402():
        enter_critical
        move_thread_flag_4402 = 1
        local towardsPos=calculate_point_to_move_towards(p[0.0,0.0,0.0,0.0,0.0,0.0], [0.0,0.0,1.0], 0.007)
        movel(towardsPos, a=0.015, v=0.015)
        move_thread_flag_4402 = 2
        exit_critical
      end
      move_thread_flag_4402 = 0
      move_thread_han_4402 = run move_thread_4402()
      while (True):
        sleep(1.0E-10)
        if (move_thread_flag_4402 > 1):
          join move_thread_han_4402
          $ 4403 "Until (distance)"
          break
        end
        sync()
      end
      $ 4404 "Wait: 0.3"
      sleep(0.3)
      $ 4405 "Set CO[1]=Encender"
      set_configurable_digital_out(1, True)
      $ 4406 "Wait: 0.3"
      sleep(0.3)
      $ 4407 "Loop 1 times"
      Loop_88 = 0
      while (Loop_88 < 1):
        $ 4408 "bajar≔pose_add(get_actual_tcp_pose(), bajada_broca)"
        global bajar= pose_add ( get_actual_tcp_pose (), bajada_broca)
        $ 4409 "bajar" "breakAfter"
        movel(bajar, a=0.004, v=0.004)
        $ 4410 "subir≔pose_sub(get_actual_tcp_pose(), bajada_broca)"
        global subir= pose_sub ( get_actual_tcp_pose (), bajada_broca)
        $ 4411 "Direction: Base Z+"
        global move_thread_flag_4411=0
        thread move_thread_4411():
          enter_critical
          move_thread_flag_4411 = 1
          local towardsPos=calculate_point_to_move_towards(p[0.0,0.0,0.0,0.0,0.0,0.0], [0.0,0.0,1.0], 0.002)
          movel(towardsPos, a=0.015, v=0.015)
          move_thread_flag_4411 = 2
          exit_critical
        end
        move_thread_flag_4411 = 0
        move_thread_han_4411 = run move_thread_4411()
        while (True):
          sleep(1.0E-10)
          if (move_thread_flag_4411 > 1):
            join move_thread_han_4411
            $ 4412 "Until (distance)"
            break
          end
